Yaskawa INFORM job: test_long_tjr3.JBI

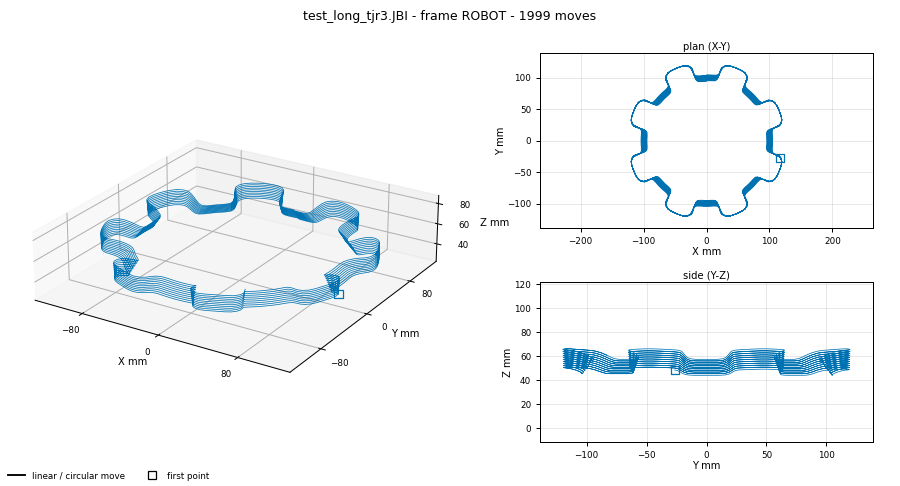
[picture p0: tool path of test_long_tjr3.JBI in frame ROBOT, 1999 of 2000 moves have a stored position in this frame; points joined in program order, loops and branches not executed]
version: 0
/JOB
//NAME test_long
//POS
///NPOS 48,0,0,2,0,0
///TOOL 1
///POSTYPE ROBOT
///RECTAN
///RCONF 1,0,0,0,0,0,0,0,0,0,0,0,0,0,0,0,0,0,0,0,0,0,0,0
C00000=118.780,-30.320,48.810,0.0300,0.0100,1.0000
C00001=116.910,-26.570,48.590,0.0400,0.0300,1.0000
C00002=114.000,-24.360,48.180,0.0300,0.0400,1.0000
C00003=110.720,-22.590,47.350,-0.0000,-0.0000,1.0000
C00004=107.770,-20.860,46.290,-0.0700,-0.1000,0.9900
C00005=105.620,-18.820,45.250,-0.2500,-0.2300,0.9400
C00006=104.550,-15.720,44.490,-0.5500,-0.1000,0.8300
C00007=104.610,-10.680,44.190,-0.6000,0.0300,0.8000
C00008=104.980,-5.420,44.180,-0.6000,0.0300,0.8000
C00009=105.130,0.000,44.190,-0.6000,0.0000,0.8000
C00010=104.980,5.420,44.180,-0.6000,-0.0300,0.8000
C00011=104.610,10.680,44.190,-0.6000,-0.0300,0.8000
C00012=104.550,15.720,44.490,-0.5500,0.1000,0.8300
C00013=105.620,18.820,45.250,-0.2500,0.2300,0.9400
C00014=107.770,20.860,46.290,-0.0700,0.1000,0.9900
C00015=110.720,22.590,47.350,-0.0000,0.0000,1.0000
C00016=114.000,24.360,48.180,0.0300,-0.0400,1.0000
C00017=116.910,26.570,48.590,0.0400,-0.0300,1.0000
C00018=118.780,30.320,48.810,0.0300,-0.0100,1.0000
C00019=119.290,35.170,48.990,0.0200,0.0000,1.0000
C00020=118.250,40.300,49.160,0.0000,0.0000,1.0000
C00021=116.480,45.340,49.280,0.0000,0.0000,1.0000
C00022=114.420,50.300,49.280,0.0000,0.0000,1.0000
C00023=112.110,55.120,49.160,0.0000,0.0000,1.0000
C00024=109.220,59.480,48.990,0.0200,0.0100,1.0000
C00025=105.430,62.550,48.810,0.0200,0.0300,1.0000
C00026=101.460,63.880,48.590,0.0000,0.0500,1.0000
C00027=97.840,63.390,48.180,-0.0100,0.0500,1.0000
C00028=94.260,62.320,47.350,0.0000,-0.0000,1.0000
C00029=90.960,61.450,46.290,0.0300,-0.1200,0.9900
C00030=87.990,61.380,45.250,-0.0200,-0.3400,0.9400
C00031=85.040,62.810,44.490,-0.3200,-0.4600,0.8300
C00032=81.530,66.420,44.190,-0.4500,-0.4000,0.8000
C00033=78.070,70.400,44.180,-0.4500,-0.4000,0.8000
C00034=74.330,74.330,44.190,-0.4300,-0.4300,0.8000
C00035=70.400,78.070,44.180,-0.4000,-0.4500,0.8000
C00036=66.420,81.530,44.190,-0.4000,-0.4500,0.8000
C00037=62.810,85.040,44.490,-0.4600,-0.3200,0.8300
C00038=61.380,87.990,45.250,-0.3400,-0.0200,0.9400
C00039=61.450,90.960,46.290,-0.1200,0.0300,0.9900
C00040=62.320,94.260,47.350,-0.0000,0.0000,1.0000
C00041=63.390,97.840,48.180,0.0500,-0.0100,1.0000
C00042=63.880,101.460,48.590,0.0500,0.0000,1.0000
C00043=62.550,105.430,48.810,0.0300,0.0200,1.0000
C00044=59.480,109.220,48.990,0.0100,0.0200,1.0000
C00045=55.120,112.110,49.160,0.0000,0.0000,1.0000
C00046=50.300,114.420,49.280,0.0000,0.0000,1.0000
C00047=45.340,116.480,49.280,0.0000,0.0000,1.0000
C00048=40.300,118.250,49.160,0.0000,0.0000,1.0000
C00049=35.170,119.290,48.990,0.0000,0.0200,1.0000
C00050=30.320,118.780,48.810,-0.0100,0.0300,1.0000
C00051=26.570,116.910,48.590,-0.0300,0.0400,1.0000
C00052=24.360,114.000,48.180,-0.0400,0.0300,1.0000
C00053=22.590,110.720,47.350,0.0000,-0.0000,1.0000
C00054=20.860,107.770,46.290,0.1000,-0.0700,0.9900
C00055=18.820,105.620,45.250,0.2300,-0.2500,0.9400
C00056=15.720,104.550,44.490,0.1000,-0.5500,0.8300
C00057=10.680,104.610,44.190,-0.0300,-0.6000,0.8000
C00058=5.420,104.980,44.180,-0.0300,-0.6000,0.8000
C00059=0.000,105.130,44.190,0.0000,-0.6000,0.8000
C00060=0.000,104.090,45.540,0.0000,-0.6100,0.7900
C00061=5.330,103.950,45.530,-0.0300,-0.6100,0.7900
C00062=10.520,103.590,45.540,-0.0300,-0.6100,0.7900
C00063=15.530,103.560,45.860,0.1100,-0.5500,0.8300
C00064=18.580,104.710,46.670,0.2300,-0.2300,0.9500
C00065=20.580,106.990,47.770,0.0900,-0.0500,0.9900
C00066=22.280,110.120,48.910,-0.0100,0.0000,1.0000
C00067=24.030,113.600,49.800,-0.0500,0.0300,1.0000
C00068=26.200,116.710,50.240,-0.0400,0.0500,1.0000
C00069=29.980,118.740,50.470,-0.0100,0.0300,1.0000
C00070=34.900,119.340,50.660,0.0000,0.0200,1.0000
C00071=40.120,118.310,50.850,0.0000,0.0000,1.0000
C00072=45.280,116.500,50.980,0.0000,0.0000,1.0000
C00073=50.360,114.400,50.980,0.0000,0.0000,1.0000
C00074=55.290,112.020,50.850,0.0000,0.0000,1.0000
C00075=59.710,109.060,50.660,0.0200,0.0200,1.0000
C00076=62.770,105.160,50.470,0.0300,0.0200,1.0000
C00077=64.000,101.050,50.240,0.0600,0.0000,1.0000
C00078=63.340,97.320,49.800,0.0600,-0.0200,1.0000
C00079=62.110,93.620,48.910,0.0100,-0.0000,1.0000
C00080=61.100,90.210,47.770,-0.1000,0.0300,0.9900
C00081=60.910,87.180,46.670,-0.3200,-0.0000,0.9500
C00082=62.250,84.200,45.860,-0.4700,-0.3100,0.8300
C00083=65.810,80.690,45.540,-0.4100,-0.4500,0.7900
C00084=69.740,77.270,45.530,-0.4100,-0.4500,0.7900
C00085=73.610,73.610,45.540,-0.4300,-0.4300,0.7900
C00086=77.270,69.740,45.530,-0.4500,-0.4100,0.7900
C00087=80.690,65.810,45.540,-0.4500,-0.4100,0.7900
C00088=84.200,62.250,45.860,-0.3100,-0.4700,0.8300
C00089=87.180,60.910,46.670,-0.0000,-0.3200,0.9500
C00090=90.210,61.100,47.770,0.0300,-0.1000,0.9900
C00091=93.620,62.110,48.910,-0.0000,0.0100,1.0000
C00092=97.320,63.340,49.800,-0.0200,0.0600,1.0000
C00093=101.050,64.000,50.240,0.0000,0.0600,1.0000
C00094=105.160,62.770,50.470,0.0200,0.0300,1.0000
C00095=109.060,59.710,50.660,0.0200,0.0200,1.0000
C00096=112.020,55.290,50.850,0.0000,0.0000,1.0000
C00097=114.400,50.360,50.980,0.0000,0.0000,1.0000
C00098=116.500,45.280,50.980,0.0000,0.0000,1.0000
C00099=118.310,40.120,50.850,0.0000,0.0000,1.0000
C00100=119.340,34.900,50.660,0.0200,0.0000,1.0000
C00101=118.740,29.980,50.470,0.0300,-0.0100,1.0000
C00102=116.710,26.200,50.240,0.0500,-0.0400,1.0000
C00103=113.600,24.030,49.800,0.0300,-0.0500,1.0000
C00104=110.120,22.280,48.910,0.0000,-0.0100,1.0000
C00105=106.990,20.580,47.770,-0.0500,0.0900,0.9900
C00106=104.710,18.580,46.670,-0.2300,0.2300,0.9500
C00107=103.560,15.530,45.860,-0.5500,0.1100,0.8300
C00108=103.590,10.520,45.540,-0.6100,-0.0300,0.7900
C00109=103.950,5.330,45.530,-0.6100,-0.0300,0.7900
C00110=104.090,0.000,45.540,-0.6100,0.0000,0.7900
C00111=103.950,-5.330,45.530,-0.6100,0.0300,0.7900
C00112=103.590,-10.520,45.540,-0.6100,0.0300,0.7900
C00113=103.560,-15.530,45.860,-0.5500,-0.1100,0.8300
C00114=104.710,-18.580,46.670,-0.2300,-0.2300,0.9500
C00115=106.990,-20.580,47.770,-0.0500,-0.0900,0.9900
C00116=110.120,-22.280,48.910,0.0000,0.0100,1.0000
C00117=113.600,-24.030,49.800,0.0300,0.0500,1.0000
C00118=116.710,-26.200,50.240,0.0500,0.0400,1.0000
C00119=118.740,-29.980,50.470,0.0300,0.0100,1.0000
C00120=119.340,-34.900,50.660,0.0200,-0.0000,1.0000
C00121=118.310,-40.120,50.850,0.0000,-0.0000,1.0000
C00122=116.500,-45.280,50.980,0.0000,-0.0000,1.0000
C00123=114.400,-50.360,50.980,0.0000,-0.0000,1.0000
C00124=112.020,-55.290,50.850,0.0000,-0.0000,1.0000
C00125=109.060,-59.710,50.660,0.0200,-0.0200,1.0000
C00126=105.160,-62.770,50.470,0.0200,-0.0300,1.0000
C00127=101.050,-64.000,50.240,0.0000,-0.0600,1.0000
C00128=97.320,-63.340,49.800,-0.0200,-0.0600,1.0000
C00129=93.620,-62.110,48.910,-0.0000,-0.0100,1.0000
C00130=90.210,-61.100,47.770,0.0300,0.1000,0.9900
C00131=87.180,-60.910,46.670,-0.0000,0.3200,0.9500
C00132=84.200,-62.250,45.860,-0.3100,0.4700,0.8300
C00133=80.690,-65.810,45.540,-0.4500,0.4100,0.7900
C00134=77.270,-69.740,45.530,-0.4500,0.4100,0.7900
C00135=73.610,-73.610,45.540,-0.4300,0.4300,0.7900
C00136=69.740,-77.270,45.530,-0.4100,0.4500,0.7900
C00137=65.810,-80.690,45.540,-0.4100,0.4500,0.7900
C00138=62.250,-84.200,45.860,-0.4700,0.3100,0.8300
C00139=60.910,-87.180,46.670,-0.3200,0.0000,0.9500
C00140=61.100,-90.210,47.770,-0.1000,-0.0300,0.9900
C00141=62.110,-93.620,48.910,0.0100,0.0000,1.0000
C00142=63.340,-97.320,49.800,0.0600,0.0200,1.0000
C00143=64.000,-101.050,50.240,0.0600,-0.0000,1.0000
C00144=62.770,-105.160,50.470,0.0300,-0.0200,1.0000
C00145=59.710,-109.060,50.660,0.0200,-0.0200,1.0000
C00146=55.290,-112.020,50.850,0.0000,-0.0000,1.0000
C00147=50.360,-114.400,50.980,0.0000,-0.0000,1.0000
C00148=45.280,-116.500,50.980,0.0000,-0.0000,1.0000
C00149=40.120,-118.310,50.850,0.0000,-0.0000,1.0000
C00150=34.900,-119.340,50.660,0.0000,-0.0200,1.0000
C00151=29.980,-118.740,50.470,-0.0100,-0.0300,1.0000
C00152=26.200,-116.710,50.240,-0.0400,-0.0500,1.0000
C00153=24.030,-113.600,49.800,-0.0500,-0.0300,1.0000
C00154=22.280,-110.120,48.910,-0.0100,-0.0000,1.0000
C00155=20.580,-106.990,47.770,0.0900,0.0500,0.9900
C00156=18.580,-104.710,46.670,0.2300,0.2300,0.9500
C00157=15.530,-103.560,45.860,0.1100,0.5500,0.8300
C00158=10.520,-103.590,45.540,-0.0300,0.6100,0.7900
C00159=5.330,-103.950,45.530,-0.0300,0.6100,0.7900
C00160=0.000,-104.090,45.540,0.0000,0.6100,0.7900
C00161=0.000,-104.090,45.540,0.0000,0.6100,0.7900
C00162=-5.330,-103.950,45.530,0.0300,0.6100,0.7900
C00163=-10.520,-103.590,45.540,0.0300,0.6100,0.7900
C00164=-15.530,-103.560,45.860,-0.1100,0.5500,0.8300
C00165=-18.580,-104.710,46.670,-0.2300,0.2300,0.9500
C00166=-20.580,-106.990,47.770,-0.0900,0.0500,0.9900
C00167=-22.280,-110.120,48.910,0.0100,-0.0000,1.0000
C00168=-24.030,-113.600,49.800,0.0500,-0.0300,1.0000
C00169=-26.200,-116.710,50.240,0.0400,-0.0500,1.0000
C00170=-29.980,-118.740,50.470,0.0100,-0.0300,1.0000
C00171=-34.900,-119.340,50.660,-0.0000,-0.0200,1.0000
C00172=-40.120,-118.310,50.850,-0.0000,-0.0000,1.0000
C00173=-45.280,-116.500,50.980,-0.0000,-0.0000,1.0000
C00174=-50.360,-114.400,50.980,-0.0000,-0.0000,1.0000
C00175=-55.290,-112.020,50.850,-0.0000,-0.0000,1.0000
C00176=-59.710,-109.060,50.660,-0.0200,-0.0200,1.0000
C00177=-62.770,-105.160,50.470,-0.0300,-0.0200,1.0000
C00178=-64.000,-101.050,50.240,-0.0600,-0.0000,1.0000
C00179=-63.340,-97.320,49.800,-0.0600,0.0200,1.0000
C00180=-62.110,-93.620,48.910,-0.0100,0.0000,1.0000
C00181=-61.100,-90.210,47.770,0.1000,-0.0300,0.9900
C00182=-60.910,-87.180,46.670,0.3200,0.0000,0.9500
C00183=-62.250,-84.200,45.860,0.4700,0.3100,0.8300
C00184=-65.810,-80.690,45.540,0.4100,0.4500,0.7900
C00185=-69.740,-77.270,45.530,0.4100,0.4500,0.7900
C00186=-73.610,-73.610,45.540,0.4300,0.4300,0.7900
C00187=-77.270,-69.740,45.530,0.4500,0.4100,0.7900
C00188=-80.690,-65.810,45.540,0.4500,0.4100,0.7900
C00189=-84.200,-62.250,45.860,0.3100,0.4700,0.8300
C00190=-87.180,-60.910,46.670,0.0000,0.3200,0.9500
C00191=-90.210,-61.100,47.770,-0.0300,0.1000,0.9900
C00192=-93.620,-62.110,48.910,0.0000,-0.0100,1.0000
C00193=-97.320,-63.340,49.800,0.0200,-0.0600,1.0000
C00194=-101.050,-64.000,50.240,-0.0000,-0.0600,1.0000
C00195=-105.160,-62.770,50.470,-0.0200,-0.0300,1.0000
C00196=-109.060,-59.710,50.660,-0.0200,-0.0200,1.0000
C00197=-112.020,-55.290,50.850,-0.0000,-0.0000,1.0000
C00198=-114.400,-50.360,50.980,-0.0000,-0.0000,1.0000
C00199=-116.500,-45.280,50.980,-0.0000,-0.0000,1.0000
C00200=-118.310,-40.120,50.850,-0.0000,-0.0000,1.0000
C00201=-119.340,-34.900,50.660,-0.0200,-0.0000,1.0000
C00202=-118.740,-29.980,50.470,-0.0300,0.0100,1.0000
C00203=-116.710,-26.200,50.240,-0.0500,0.0400,1.0000
C00204=-113.600,-24.030,49.800,-0.0300,0.0500,1.0000
C00205=-110.120,-22.280,48.910,-0.0000,0.0100,1.0000
C00206=-106.990,-20.580,47.770,0.0500,-0.0900,0.9900
C00207=-104.710,-18.580,46.670,0.2300,-0.2300,0.9500
C00208=-103.560,-15.530,45.860,0.5500,-0.1100,0.8300
C00209=-103.590,-10.520,45.540,0.6100,0.0300,0.7900
C00210=-103.950,-5.330,45.530,0.6100,0.0300,0.7900
C00211=-104.090,0.000,45.540,0.6100,-0.0000,0.7900
C00212=-103.950,5.330,45.530,0.6100,-0.0300,0.7900
C00213=-103.590,10.520,45.540,0.6100,-0.0300,0.7900
C00214=-103.560,15.530,45.860,0.5500,0.1100,0.8300
C00215=-104.710,18.580,46.670,0.2300,0.2300,0.9500
C00216=-106.990,20.580,47.770,0.0500,0.0900,0.9900
C00217=-110.120,22.280,48.910,-0.0000,-0.0100,1.0000
C00218=-113.600,24.030,49.800,-0.0300,-0.0500,1.0000
C00219=-116.710,26.200,50.240,-0.0500,-0.0400,1.0000
C00220=-118.740,29.980,50.470,-0.0300,-0.0100,1.0000
C00221=-119.340,34.900,50.660,-0.0200,0.0000,1.0000
C00222=-118.310,40.120,50.850,-0.0000,0.0000,1.0000
C00223=-116.500,45.280,50.980,-0.0000,0.0000,1.0000
C00224=-114.400,50.360,50.980,-0.0000,0.0000,1.0000
C00225=-112.020,55.290,50.850,-0.0000,0.0000,1.0000
C00226=-109.060,59.710,50.660,-0.0200,0.0200,1.0000
C00227=-105.160,62.770,50.470,-0.0200,0.0300,1.0000
C00228=-101.050,64.000,50.240,-0.0000,0.0600,1.0000
C00229=-97.320,63.340,49.800,0.0200,0.0600,1.0000
C00230=-93.620,62.110,48.910,0.0000,0.0100,1.0000
C00231=-90.210,61.100,47.770,-0.0300,-0.1000,0.9900
C00232=-87.180,60.910,46.670,0.0000,-0.3200,0.9500
C00233=-84.200,62.250,45.860,0.3100,-0.4700,0.8300
C00234=-80.690,65.810,45.540,0.4500,-0.4100,0.7900
C00235=-77.270,69.740,45.530,0.4500,-0.4100,0.7900
C00236=-73.610,73.610,45.540,0.4300,-0.4300,0.7900
C00237=-69.740,77.270,45.530,0.4100,-0.4500,0.7900
C00238=-65.810,80.690,45.540,0.4100,-0.4500,0.7900
C00239=-62.250,84.200,45.860,0.4700,-0.3100,0.8300
C00240=-60.910,87.180,46.670,0.3200,-0.0000,0.9500
C00241=-61.100,90.210,47.770,0.1000,0.0300,0.9900
C00242=-62.110,93.620,48.910,-0.0100,-0.0000,1.0000
C00243=-63.340,97.320,49.800,-0.0600,-0.0200,1.0000
C00244=-64.000,101.050,50.240,-0.0600,0.0000,1.0000
C00245=-62.770,105.160,50.470,-0.0300,0.0200,1.0000
C00246=-59.710,109.060,50.660,-0.0200,0.0200,1.0000
C00247=-55.290,112.020,50.850,-0.0000,0.0000,1.0000
C00248=-50.360,114.400,50.980,-0.0000,0.0000,1.0000
C00249=-45.280,116.500,50.980,-0.0000,0.0000,1.0000
C00250=-40.120,118.310,50.850,-0.0000,0.0000,1.0000
C00251=-34.900,119.340,50.660,-0.0000,0.0200,1.0000
C00252=-29.980,118.740,50.470,0.0100,0.0300,1.0000
C00253=-26.200,116.710,50.240,0.0400,0.0500,1.0000
C00254=-24.030,113.600,49.800,0.0500,0.0300,1.0000
C00255=-22.280,110.120,48.910,0.0100,0.0000,1.0000
C00256=-20.580,106.990,47.770,-0.0900,-0.0500,0.9900
C00257=-18.580,104.710,46.670,-0.2300,-0.2300,0.9500
C00258=-15.530,103.560,45.860,-0.1100,-0.5500,0.8300
C00259=-10.520,103.590,45.540,0.0300,-0.6100,0.7900
C00260=-5.330,103.950,45.530,0.0300,-0.6100,0.7900
C00261=0.000,104.090,45.540,0.0000,-0.6100,0.7900
C00262=0.000,103.050,46.880,0.0000,-0.6100,0.7900
C00263=-5.230,102.920,46.870,0.0300,-0.6100,0.7900
C00264=-10.360,102.570,46.890,0.0300,-0.6100,0.7900
C00265=-15.330,102.560,47.230,-0.1200,-0.5500,0.8200
C00266=-18.330,103.800,48.080,-0.2200,-0.2100,0.9500
C00267=-20.300,106.210,49.250,-0.0800,-0.0400,1.0000
C00268=-21.970,109.510,50.470,0.0200,0.0100,1.0000
C00269=-23.690,113.200,51.410,0.0600,0.0300,1.0000
C00270=-25.830,116.510,51.880,0.0500,0.0500,1.0000
C00271=-29.630,118.700,52.130,0.0100,0.0400,1.0000
C00272=-34.620,119.390,52.340,-0.0000,0.0300,1.0000
C00273=-39.940,118.360,52.540,-0.0000,0.0000,1.0000
C00274=-45.220,116.520,52.680,-0.0000,0.0000,1.0000
C00275=-50.420,114.370,52.680,-0.0000,0.0000,1.0000
C00276=-55.450,111.940,52.540,-0.0000,0.0000,1.0000
C00277=-59.940,108.900,52.340,-0.0200,0.0200,1.0000
C00278=-62.980,104.880,52.130,-0.0400,0.0200,1.0000
C00279=-64.120,100.650,51.880,-0.0700,0.0000,1.0000
C00280=-63.290,96.790,51.410,-0.0700,-0.0200,1.0000
C00281=-61.900,92.970,50.470,-0.0200,-0.0100,1.0000
C00282=-60.750,89.460,49.250,0.0900,0.0200,1.0000
C00283=-60.430,86.360,48.080,0.3100,0.0100,0.9500
C00284=-61.680,83.360,47.230,0.4800,-0.3100,0.8200
C00285=-65.200,79.850,46.890,0.4100,-0.4500,0.7900
C00286=-69.070,76.470,46.870,0.4100,-0.4600,0.7900
C00287=-72.870,72.870,46.880,0.4300,-0.4300,0.7900
C00288=-76.470,69.070,46.870,0.4600,-0.4100,0.7900
C00289=-79.850,65.200,46.890,0.4500,-0.4100,0.7900
C00290=-83.360,61.680,47.230,0.3100,-0.4800,0.8200
C00291=-86.360,60.430,48.080,-0.0100,-0.3100,0.9500
C00292=-89.460,60.750,49.250,-0.0200,-0.0900,1.0000
C00293=-92.970,61.900,50.470,0.0100,0.0200,1.0000
C00294=-96.790,63.290,51.410,0.0200,0.0700,1.0000
C00295=-100.650,64.120,51.880,-0.0000,0.0700,1.0000
C00296=-104.880,62.980,52.130,-0.0200,0.0400,1.0000
C00297=-108.900,59.940,52.340,-0.0200,0.0200,1.0000
C00298=-111.940,55.450,52.540,-0.0000,0.0000,1.0000
C00299=-114.370,50.420,52.680,-0.0000,0.0000,1.0000
C00300=-116.520,45.220,52.680,-0.0000,0.0000,1.0000
C00301=-118.360,39.940,52.540,-0.0000,0.0000,1.0000
C00302=-119.390,34.620,52.340,-0.0300,0.0000,1.0000
C00303=-118.700,29.630,52.130,-0.0400,-0.0100,1.0000
C00304=-116.510,25.830,51.880,-0.0500,-0.0500,1.0000
C00305=-113.200,23.690,51.410,-0.0300,-0.0600,1.0000
C00306=-109.510,21.970,50.470,-0.0100,-0.0200,1.0000
C00307=-106.210,20.300,49.250,0.0400,0.0800,1.0000
C00308=-103.800,18.330,48.080,0.2100,0.2200,0.9500
C00309=-102.560,15.330,47.230,0.5500,0.1200,0.8200
C00310=-102.570,10.360,46.890,0.6100,-0.0300,0.7900
C00311=-102.920,5.230,46.870,0.6100,-0.0300,0.7900
C00312=-103.050,0.000,46.880,0.6100,-0.0000,0.7900
C00313=-102.920,-5.230,46.870,0.6100,0.0300,0.7900
C00314=-102.570,-10.360,46.890,0.6100,0.0300,0.7900
C00315=-102.560,-15.330,47.230,0.5500,-0.1200,0.8200
C00316=-103.800,-18.330,48.080,0.2100,-0.2200,0.9500
C00317=-106.210,-20.300,49.250,0.0400,-0.0800,1.0000
C00318=-109.510,-21.970,50.470,-0.0100,0.0200,1.0000
C00319=-113.200,-23.690,51.410,-0.0300,0.0600,1.0000
C00320=-116.510,-25.830,51.880,-0.0500,0.0500,1.0000
C00321=-118.700,-29.630,52.130,-0.0400,0.0100,1.0000
C00322=-119.390,-34.620,52.340,-0.0300,-0.0000,1.0000
C00323=-118.360,-39.940,52.540,-0.0000,-0.0000,1.0000
C00324=-116.520,-45.220,52.680,-0.0000,-0.0000,1.0000
C00325=-114.370,-50.420,52.680,-0.0000,-0.0000,1.0000
C00326=-111.940,-55.450,52.540,-0.0000,-0.0000,1.0000
C00327=-108.900,-59.940,52.340,-0.0200,-0.0200,1.0000
C00328=-104.880,-62.980,52.130,-0.0200,-0.0400,1.0000
C00329=-100.650,-64.120,51.880,-0.0000,-0.0700,1.0000
C00330=-96.790,-63.290,51.410,0.0200,-0.0700,1.0000
C00331=-92.970,-61.900,50.470,0.0100,-0.0200,1.0000
C00332=-89.460,-60.750,49.250,-0.0200,0.0900,1.0000
C00333=-86.360,-60.430,48.080,-0.0100,0.3100,0.9500
C00334=-83.360,-61.680,47.230,0.3100,0.4800,0.8200
C00335=-79.850,-65.200,46.890,0.4500,0.4100,0.7900
C00336=-76.470,-69.070,46.870,0.4600,0.4100,0.7900
C00337=-72.870,-72.870,46.880,0.4300,0.4300,0.7900
C00338=-69.070,-76.470,46.870,0.4100,0.4600,0.7900
C00339=-65.200,-79.850,46.890,0.4100,0.4500,0.7900
C00340=-61.680,-83.360,47.230,0.4800,0.3100,0.8200
C00341=-60.430,-86.360,48.080,0.3100,-0.0100,0.9500
C00342=-60.750,-89.460,49.250,0.0900,-0.0200,1.0000
C00343=-61.900,-92.970,50.470,-0.0200,0.0100,1.0000
C00344=-63.290,-96.790,51.410,-0.0700,0.0200,1.0000
C00345=-64.120,-100.650,51.880,-0.0700,-0.0000,1.0000
C00346=-62.980,-104.880,52.130,-0.0400,-0.0200,1.0000
C00347=-59.940,-108.900,52.340,-0.0200,-0.0200,1.0000
C00348=-55.450,-111.940,52.540,-0.0000,-0.0000,1.0000
C00349=-50.420,-114.370,52.680,-0.0000,-0.0000,1.0000
C00350=-45.220,-116.520,52.680,-0.0000,-0.0000,1.0000
C00351=-39.940,-118.360,52.540,-0.0000,-0.0000,1.0000
C00352=-34.620,-119.390,52.340,-0.0000,-0.0300,1.0000
C00353=-29.630,-118.700,52.130,0.0100,-0.0400,1.0000
C00354=-25.830,-116.510,51.880,0.0500,-0.0500,1.0000
C00355=-23.690,-113.200,51.410,0.0600,-0.0300,1.0000
C00356=-21.970,-109.510,50.470,0.0200,-0.0100,1.0000
C00357=-20.300,-106.210,49.250,-0.0800,0.0400,1.0000
C00358=-18.330,-103.800,48.080,-0.2200,0.2100,0.9500
C00359=-15.330,-102.560,47.230,-0.1200,0.5500,0.8200
C00360=-10.360,-102.570,46.890,0.0300,0.6100,0.7900
C00361=-5.230,-102.920,46.870,0.0300,0.6100,0.7900
C00362=0.000,-103.050,46.880,0.0000,0.6100,0.7900
C00363=0.000,-103.050,46.880,0.0000,0.6100,0.7900
C00364=5.230,-102.920,46.870,-0.0300,0.6100,0.7900
C00365=10.360,-102.570,46.890,-0.0300,0.6100,0.7900
C00366=15.330,-102.560,47.230,0.1200,0.5500,0.8200
C00367=18.330,-103.800,48.080,0.2200,0.2100,0.9500
C00368=20.300,-106.210,49.250,0.0800,0.0400,1.0000
C00369=21.970,-109.510,50.470,-0.0200,-0.0100,1.0000
C00370=23.690,-113.200,51.410,-0.0600,-0.0300,1.0000
C00371=25.830,-116.510,51.880,-0.0500,-0.0500,1.0000
C00372=29.630,-118.700,52.130,-0.0100,-0.0400,1.0000
C00373=34.620,-119.390,52.340,0.0000,-0.0300,1.0000
C00374=39.940,-118.360,52.540,0.0000,-0.0000,1.0000
C00375=45.220,-116.520,52.680,0.0000,-0.0000,1.0000
C00376=50.420,-114.370,52.680,0.0000,-0.0000,1.0000
C00377=55.450,-111.940,52.540,0.0000,-0.0000,1.0000
C00378=59.940,-108.900,52.340,0.0200,-0.0200,1.0000
C00379=62.980,-104.880,52.130,0.0400,-0.0200,1.0000
C00380=64.120,-100.650,51.880,0.0700,-0.0000,1.0000
C00381=63.290,-96.790,51.410,0.0700,0.0200,1.0000
C00382=61.900,-92.970,50.470,0.0200,0.0100,1.0000
C00383=60.750,-89.460,49.250,-0.0900,-0.0200,1.0000
C00384=60.430,-86.360,48.080,-0.3100,-0.0100,0.9500
C00385=61.680,-83.360,47.230,-0.4800,0.3100,0.8200
C00386=65.200,-79.850,46.890,-0.4100,0.4500,0.7900
C00387=69.070,-76.470,46.870,-0.4100,0.4600,0.7900
C00388=72.870,-72.870,46.880,-0.4300,0.4300,0.7900
C00389=76.470,-69.070,46.870,-0.4600,0.4100,0.7900
C00390=79.850,-65.200,46.890,-0.4500,0.4100,0.7900
C00391=83.360,-61.680,47.230,-0.3100,0.4800,0.8200
C00392=86.360,-60.430,48.080,0.0100,0.3100,0.9500
C00393=89.460,-60.750,49.250,0.0200,0.0900,1.0000
C00394=92.970,-61.900,50.470,-0.0100,-0.0200,1.0000
C00395=96.790,-63.290,51.410,-0.0200,-0.0700,1.0000
C00396=100.650,-64.120,51.880,0.0000,-0.0700,1.0000
C00397=104.880,-62.980,52.130,0.0200,-0.0400,1.0000
C00398=108.900,-59.940,52.340,0.0200,-0.0200,1.0000
C00399=111.940,-55.450,52.540,0.0000,-0.0000,1.0000
C00400=114.370,-50.420,52.680,0.0000,-0.0000,1.0000
C00401=116.520,-45.220,52.680,0.0000,-0.0000,1.0000
C00402=118.360,-39.940,52.540,0.0000,-0.0000,1.0000
C00403=119.390,-34.620,52.340,0.0300,-0.0000,1.0000
C00404=118.700,-29.630,52.130,0.0400,0.0100,1.0000
C00405=116.510,-25.830,51.880,0.0500,0.0500,1.0000
C00406=113.200,-23.690,51.410,0.0300,0.0600,1.0000
C00407=109.510,-21.970,50.470,0.0100,0.0200,1.0000
C00408=106.210,-20.300,49.250,-0.0400,-0.0800,1.0000
C00409=103.800,-18.330,48.080,-0.2100,-0.2200,0.9500
C00410=102.560,-15.330,47.230,-0.5500,-0.1200,0.8200
C00411=102.570,-10.360,46.890,-0.6100,0.0300,0.7900
C00412=102.920,-5.230,46.870,-0.6100,0.0300,0.7900
C00413=103.050,0.000,46.880,-0.6100,0.0000,0.7900
C00414=102.920,5.230,46.870,-0.6100,-0.0300,0.7900
C00415=102.570,10.360,46.890,-0.6100,-0.0300,0.7900
C00416=102.560,15.330,47.230,-0.5500,0.1200,0.8200
C00417=103.800,18.330,48.080,-0.2100,0.2200,0.9500
C00418=106.210,20.300,49.250,-0.0400,0.0800,1.0000
C00419=109.510,21.970,50.470,0.0100,-0.0200,1.0000
C00420=113.200,23.690,51.410,0.0300,-0.0600,1.0000
C00421=116.510,25.830,51.880,0.0500,-0.0500,1.0000
C00422=118.700,29.630,52.130,0.0400,-0.0100,1.0000
C00423=119.390,34.620,52.340,0.0300,0.0000,1.0000
C00424=118.360,39.940,52.540,0.0000,0.0000,1.0000
C00425=116.520,45.220,52.680,0.0000,0.0000,1.0000
C00426=114.370,50.420,52.680,0.0000,0.0000,1.0000
C00427=111.940,55.450,52.540,0.0000,0.0000,1.0000
C00428=108.900,59.940,52.340,0.0200,0.0200,1.0000
C00429=104.880,62.980,52.130,0.0200,0.0400,1.0000
C00430=100.650,64.120,51.880,0.0000,0.0700,1.0000
C00431=96.790,63.290,51.410,-0.0200,0.0700,1.0000
C00432=92.970,61.900,50.470,-0.0100,0.0200,1.0000
C00433=89.460,60.750,49.250,0.0200,-0.0900,1.0000
C00434=86.360,60.430,48.080,0.0100,-0.3100,0.9500
C00435=83.360,61.680,47.230,-0.3100,-0.4800,0.8200
C00436=79.850,65.200,46.890,-0.4500,-0.4100,0.7900
C00437=76.470,69.070,46.870,-0.4600,-0.4100,0.7900
C00438=72.870,72.870,46.880,-0.4300,-0.4300,0.7900
C00439=69.070,76.470,46.870,-0.4100,-0.4600,0.7900
C00440=65.200,79.850,46.890,-0.4100,-0.4500,0.7900
C00441=61.680,83.360,47.230,-0.4800,-0.3100,0.8200
C00442=60.430,86.360,48.080,-0.3100,0.0100,0.9500
C00443=60.750,89.460,49.250,-0.0900,0.0200,1.0000
C00444=61.900,92.970,50.470,0.0200,-0.0100,1.0000
C00445=63.290,96.790,51.410,0.0700,-0.0200,1.0000
C00446=64.120,100.650,51.880,0.0700,0.0000,1.0000
C00447=62.980,104.880,52.130,0.0400,0.0200,1.0000
C00448=59.940,108.900,52.340,0.0200,0.0200,1.0000
C00449=55.450,111.940,52.540,0.0000,0.0000,1.0000
C00450=50.420,114.370,52.680,0.0000,0.0000,1.0000
C00451=45.220,116.520,52.680,0.0000,0.0000,1.0000
C00452=39.940,118.360,52.540,0.0000,0.0000,1.0000
C00453=34.620,119.390,52.340,0.0000,0.0300,1.0000
C00454=29.630,118.700,52.130,-0.0100,0.0400,1.0000
C00455=25.830,116.510,51.880,-0.0500,0.0500,1.0000
C00456=23.690,113.200,51.410,-0.0600,0.0300,1.0000
C00457=21.970,109.510,50.470,-0.0200,0.0100,1.0000
C00458=20.300,106.210,49.250,0.0800,-0.0400,1.0000
C00459=18.330,103.800,48.080,0.2200,-0.2100,0.9500
C00460=15.330,102.560,47.230,0.1200,-0.5500,0.8200
C00461=10.360,102.570,46.890,-0.0300,-0.6100,0.7900
C00462=5.230,102.920,46.870,-0.0300,-0.6100,0.7900
C00463=0.000,103.050,46.880,0.0000,-0.6100,0.7900
C00464=0.000,102.010,48.220,0.0000,-0.6200,0.7900
C00465=5.140,101.870,48.210,-0.0300,-0.6200,0.7900
C00466=10.200,101.530,48.230,-0.0300,-0.6100,0.7900
C00467=15.130,101.560,48.590,0.1300,-0.5500,0.8200
C00468=18.090,102.880,49.490,0.2200,-0.1900,0.9600
C00469=20.020,105.420,50.730,0.0700,-0.0400,1.0000
C00470=21.650,108.900,52.030,-0.0300,0.0100,1.0000
C00471=23.350,112.790,53.030,-0.0700,0.0300,1.0000
C00472=25.460,116.310,53.530,-0.0600,0.0500,1.0000
C00473=29.270,118.660,53.800,-0.0100,0.0400,1.0000
C00474=34.340,119.440,54.010,0.0000,0.0300,1.0000
C00475=39.770,118.420,54.230,0.0000,0.0000,1.0000
C00476=45.160,116.550,54.380,0.0000,0.0000,1.0000
C00477=50.480,114.340,54.380,0.0000,0.0000,1.0000
C00478=55.620,111.860,54.230,0.0000,0.0000,1.0000
C00479=60.180,108.740,54.010,0.0200,0.0200,1.0000
C00480=63.200,104.600,53.800,0.0400,0.0200,1.0000
C00481=64.240,100.240,53.530,0.0800,-0.0000,1.0000
C00482=63.250,96.260,53.030,0.0800,-0.0300,1.0000
C00483=61.690,92.310,52.030,0.0300,-0.0100,1.0000
C00484=60.390,88.700,50.730,-0.0700,0.0200,1.0000
C00485=59.950,85.540,49.490,-0.2900,0.0200,0.9600
C00486=61.110,82.510,48.590,-0.4800,-0.3000,0.8200
C00487=64.580,79.010,48.230,-0.4200,-0.4500,0.7900
C00488=68.400,75.670,48.210,-0.4100,-0.4600,0.7900
C00489=72.130,72.130,48.220,-0.4400,-0.4400,0.7900
C00490=75.670,68.400,48.210,-0.4600,-0.4100,0.7900
C00491=79.010,64.580,48.230,-0.4500,-0.4200,0.7900
C00492=82.510,61.110,48.590,-0.3000,-0.4800,0.8200
C00493=85.540,59.950,49.490,0.0200,-0.2900,0.9600
C00494=88.700,60.390,50.730,0.0200,-0.0700,1.0000
C00495=92.310,61.690,52.030,-0.0100,0.0300,1.0000
C00496=96.260,63.250,53.030,-0.0300,0.0800,1.0000
C00497=100.240,64.240,53.530,-0.0000,0.0800,1.0000
C00498=104.600,63.200,53.800,0.0200,0.0400,1.0000
C00499=108.740,60.180,54.010,0.0200,0.0200,1.0000
C00500=111.860,55.620,54.230,0.0000,0.0000,1.0000
C00501=114.340,50.480,54.380,0.0000,0.0000,1.0000
C00502=116.550,45.160,54.380,0.0000,0.0000,1.0000
C00503=118.420,39.770,54.230,0.0000,0.0000,1.0000
C00504=119.440,34.340,54.010,0.0300,0.0000,1.0000
C00505=118.660,29.270,53.800,0.0400,-0.0100,1.0000
C00506=116.310,25.460,53.530,0.0500,-0.0600,1.0000
C00507=112.790,23.350,53.030,0.0300,-0.0700,1.0000
C00508=108.900,21.650,52.030,0.0100,-0.0300,1.0000
C00509=105.420,20.020,50.730,-0.0400,0.0700,1.0000
C00510=102.880,18.090,49.490,-0.1900,0.2200,0.9600
C00511=101.560,15.130,48.590,-0.5500,0.1300,0.8200
C00512=101.530,10.200,48.230,-0.6100,-0.0300,0.7900
C00513=101.870,5.140,48.210,-0.6200,-0.0300,0.7900
C00514=102.010,0.000,48.220,-0.6200,0.0000,0.7900
C00515=101.870,-5.140,48.210,-0.6200,0.0300,0.7900
C00516=101.530,-10.200,48.230,-0.6100,0.0300,0.7900
C00517=101.560,-15.130,48.590,-0.5500,-0.1300,0.8200
C00518=102.880,-18.090,49.490,-0.1900,-0.2200,0.9600
C00519=105.420,-20.020,50.730,-0.0400,-0.0700,1.0000
C00520=108.900,-21.650,52.030,0.0100,0.0300,1.0000
C00521=112.790,-23.350,53.030,0.0300,0.0700,1.0000
C00522=116.310,-25.460,53.530,0.0500,0.0600,1.0000
C00523=118.660,-29.270,53.800,0.0400,0.0100,1.0000
C00524=119.440,-34.340,54.010,0.0300,-0.0000,1.0000
C00525=118.420,-39.770,54.230,0.0000,-0.0000,1.0000
C00526=116.550,-45.160,54.380,0.0000,-0.0000,1.0000
C00527=114.340,-50.480,54.380,0.0000,-0.0000,1.0000
C00528=111.860,-55.620,54.230,0.0000,-0.0000,1.0000
C00529=108.740,-60.180,54.010,0.0200,-0.0200,1.0000
C00530=104.600,-63.200,53.800,0.0200,-0.0400,1.0000
C00531=100.240,-64.240,53.530,-0.0000,-0.0800,1.0000
C00532=96.260,-63.250,53.030,-0.0300,-0.0800,1.0000
C00533=92.310,-61.690,52.030,-0.0100,-0.0300,1.0000
C00534=88.700,-60.390,50.730,0.0200,0.0700,1.0000
C00535=85.540,-59.950,49.490,0.0200,0.2900,0.9600
C00536=82.510,-61.110,48.590,-0.3000,0.4800,0.8200
C00537=79.010,-64.580,48.230,-0.4500,0.4200,0.7900
C00538=75.670,-68.400,48.210,-0.4600,0.4100,0.7900
C00539=72.130,-72.130,48.220,-0.4400,0.4400,0.7900
C00540=68.400,-75.670,48.210,-0.4100,0.4600,0.7900
C00541=64.580,-79.010,48.230,-0.4200,0.4500,0.7900
C00542=61.110,-82.510,48.590,-0.4800,0.3000,0.8200
C00543=59.950,-85.540,49.490,-0.2900,-0.0200,0.9600
C00544=60.390,-88.700,50.730,-0.0700,-0.0200,1.0000
C00545=61.690,-92.310,52.030,0.0300,0.0100,1.0000
C00546=63.250,-96.260,53.030,0.0800,0.0300,1.0000
C00547=64.240,-100.240,53.530,0.0800,0.0000,1.0000
C00548=63.200,-104.600,53.800,0.0400,-0.0200,1.0000
C00549=60.180,-108.740,54.010,0.0200,-0.0200,1.0000
C00550=55.620,-111.860,54.230,0.0000,-0.0000,1.0000
C00551=50.480,-114.340,54.380,0.0000,-0.0000,1.0000
C00552=45.160,-116.550,54.380,0.0000,-0.0000,1.0000
C00553=39.770,-118.420,54.230,0.0000,-0.0000,1.0000
C00554=34.340,-119.440,54.010,0.0000,-0.0300,1.0000
C00555=29.270,-118.660,53.800,-0.0100,-0.0400,1.0000
C00556=25.460,-116.310,53.530,-0.0600,-0.0500,1.0000
C00557=23.350,-112.790,53.030,-0.0700,-0.0300,1.0000
C00558=21.650,-108.900,52.030,-0.0300,-0.0100,1.0000
C00559=20.020,-105.420,50.730,0.0700,0.0400,1.0000
C00560=18.090,-102.880,49.490,0.2200,0.1900,0.9600
C00561=15.130,-101.560,48.590,0.1300,0.5500,0.8200
C00562=10.200,-101.530,48.230,-0.0300,0.6100,0.7900
C00563=5.140,-101.870,48.210,-0.0300,0.6200,0.7900
C00564=0.000,-102.010,48.220,0.0000,0.6200,0.7900
C00565=0.000,-102.010,48.220,0.0000,0.6200,0.7900
C00566=-5.140,-101.870,48.210,0.0300,0.6200,0.7900
C00567=-10.200,-101.530,48.230,0.0300,0.6100,0.7900
C00568=-15.130,-101.560,48.590,-0.1300,0.5500,0.8200
C00569=-18.090,-102.880,49.490,-0.2200,0.1900,0.9600
C00570=-20.020,-105.420,50.730,-0.0700,0.0400,1.0000
C00571=-21.650,-108.900,52.030,0.0300,-0.0100,1.0000
C00572=-23.350,-112.790,53.030,0.0700,-0.0300,1.0000
C00573=-25.460,-116.310,53.530,0.0600,-0.0500,1.0000
C00574=-29.270,-118.660,53.800,0.0100,-0.0400,1.0000
C00575=-34.340,-119.440,54.010,-0.0000,-0.0300,1.0000
C00576=-39.770,-118.420,54.230,-0.0000,-0.0000,1.0000
C00577=-45.160,-116.550,54.380,-0.0000,-0.0000,1.0000
C00578=-50.480,-114.340,54.380,-0.0000,-0.0000,1.0000
C00579=-55.620,-111.860,54.230,-0.0000,-0.0000,1.0000
C00580=-60.180,-108.740,54.010,-0.0200,-0.0200,1.0000
C00581=-63.200,-104.600,53.800,-0.0400,-0.0200,1.0000
C00582=-64.240,-100.240,53.530,-0.0800,0.0000,1.0000
C00583=-63.250,-96.260,53.030,-0.0800,0.0300,1.0000
C00584=-61.690,-92.310,52.030,-0.0300,0.0100,1.0000
C00585=-60.390,-88.700,50.730,0.0700,-0.0200,1.0000
C00586=-59.950,-85.540,49.490,0.2900,-0.0200,0.9600
C00587=-61.110,-82.510,48.590,0.4800,0.3000,0.8200
C00588=-64.580,-79.010,48.230,0.4200,0.4500,0.7900
C00589=-68.400,-75.670,48.210,0.4100,0.4600,0.7900
C00590=-72.130,-72.130,48.220,0.4400,0.4400,0.7900
C00591=-75.670,-68.400,48.210,0.4600,0.4100,0.7900
C00592=-79.010,-64.580,48.230,0.4500,0.4200,0.7900
C00593=-82.510,-61.110,48.590,0.3000,0.4800,0.8200
C00594=-85.540,-59.950,49.490,-0.0200,0.2900,0.9600
C00595=-88.700,-60.390,50.730,-0.0200,0.0700,1.0000
C00596=-92.310,-61.690,52.030,0.0100,-0.0300,1.0000
C00597=-96.260,-63.250,53.030,0.0300,-0.0800,1.0000
C00598=-100.240,-64.240,53.530,0.0000,-0.0800,1.0000
C00599=-104.600,-63.200,53.800,-0.0200,-0.0400,1.0000
C00600=-108.740,-60.180,54.010,-0.0200,-0.0200,1.0000
C00601=-111.860,-55.620,54.230,-0.0000,-0.0000,1.0000
C00602=-114.340,-50.480,54.380,-0.0000,-0.0000,1.0000
C00603=-116.550,-45.160,54.380,-0.0000,-0.0000,1.0000
C00604=-118.420,-39.770,54.230,-0.0000,-0.0000,1.0000
C00605=-119.440,-34.340,54.010,-0.0300,-0.0000,1.0000
C00606=-118.660,-29.270,53.800,-0.0400,0.0100,1.0000
C00607=-116.310,-25.460,53.530,-0.0500,0.0600,1.0000
C00608=-112.790,-23.350,53.030,-0.0300,0.0700,1.0000
C00609=-108.900,-21.650,52.030,-0.0100,0.0300,1.0000
C00610=-105.420,-20.020,50.730,0.0400,-0.0700,1.0000
C00611=-102.880,-18.090,49.490,0.1900,-0.2200,0.9600
C00612=-101.560,-15.130,48.590,0.5500,-0.1300,0.8200
C00613=-101.530,-10.200,48.230,0.6100,0.0300,0.7900
C00614=-101.870,-5.140,48.210,0.6200,0.0300,0.7900
C00615=-102.010,0.000,48.220,0.6200,-0.0000,0.7900
C00616=-101.870,5.140,48.210,0.6200,-0.0300,0.7900
C00617=-101.530,10.200,48.230,0.6100,-0.0300,0.7900
C00618=-101.560,15.130,48.590,0.5500,0.1300,0.8200
C00619=-102.880,18.090,49.490,0.1900,0.2200,0.9600
C00620=-105.420,20.020,50.730,0.0400,0.0700,1.0000
C00621=-108.900,21.650,52.030,-0.0100,-0.0300,1.0000
C00622=-112.790,23.350,53.030,-0.0300,-0.0700,1.0000
C00623=-116.310,25.460,53.530,-0.0500,-0.0600,1.0000
C00624=-118.660,29.270,53.800,-0.0400,-0.0100,1.0000
C00625=-119.440,34.340,54.010,-0.0300,0.0000,1.0000
C00626=-118.420,39.770,54.230,-0.0000,0.0000,1.0000
C00627=-116.550,45.160,54.380,-0.0000,0.0000,1.0000
C00628=-114.340,50.480,54.380,-0.0000,0.0000,1.0000
C00629=-111.860,55.620,54.230,-0.0000,0.0000,1.0000
C00630=-108.740,60.180,54.010,-0.0200,0.0200,1.0000
C00631=-104.600,63.200,53.800,-0.0200,0.0400,1.0000
C00632=-100.240,64.240,53.530,0.0000,0.0800,1.0000
C00633=-96.260,63.250,53.030,0.0300,0.0800,1.0000
C00634=-92.310,61.690,52.030,0.0100,0.0300,1.0000
C00635=-88.700,60.390,50.730,-0.0200,-0.0700,1.0000
C00636=-85.540,59.950,49.490,-0.0200,-0.2900,0.9600
C00637=-82.510,61.110,48.590,0.3000,-0.4800,0.8200
C00638=-79.010,64.580,48.230,0.4500,-0.4200,0.7900
C00639=-75.670,68.400,48.210,0.4600,-0.4100,0.7900
C00640=-72.130,72.130,48.220,0.4400,-0.4400,0.7900
C00641=-68.400,75.670,48.210,0.4100,-0.4600,0.7900
C00642=-64.580,79.010,48.230,0.4200,-0.4500,0.7900
C00643=-61.110,82.510,48.590,0.4800,-0.3000,0.8200
C00644=-59.950,85.540,49.490,0.2900,0.0200,0.9600
C00645=-60.390,88.700,50.730,0.0700,0.0200,1.0000
C00646=-61.690,92.310,52.030,-0.0300,-0.0100,1.0000
C00647=-63.250,96.260,53.030,-0.0800,-0.0300,1.0000
C00648=-64.240,100.240,53.530,-0.0800,-0.0000,1.0000
C00649=-63.200,104.600,53.800,-0.0400,0.0200,1.0000
C00650=-60.180,108.740,54.010,-0.0200,0.0200,1.0000
C00651=-55.620,111.860,54.230,-0.0000,0.0000,1.0000
C00652=-50.480,114.340,54.380,-0.0000,0.0000,1.0000
C00653=-45.160,116.550,54.380,-0.0000,0.0000,1.0000
C00654=-39.770,118.420,54.230,-0.0000,0.0000,1.0000
C00655=-34.340,119.440,54.010,-0.0000,0.0300,1.0000
C00656=-29.270,118.660,53.800,0.0100,0.0400,1.0000
C00657=-25.460,116.310,53.530,0.0600,0.0500,1.0000
C00658=-23.350,112.790,53.030,0.0700,0.0300,1.0000
C00659=-21.650,108.900,52.030,0.0300,0.0100,1.0000
C00660=-20.020,105.420,50.730,-0.0700,-0.0400,1.0000
C00661=-18.090,102.880,49.490,-0.2200,-0.1900,0.9600
C00662=-15.130,101.560,48.590,-0.1300,-0.5500,0.8200
C00663=-10.200,101.530,48.230,0.0300,-0.6100,0.7900
C00664=-5.140,101.870,48.210,0.0300,-0.6200,0.7900
C00665=0.000,102.010,48.220,0.0000,-0.6200,0.7900
C00666=0.000,100.950,49.560,0.0000,-0.6200,0.7800
C00667=-5.040,100.820,49.550,0.0300,-0.6200,0.7800
C00668=-10.040,100.490,49.560,0.0200,-0.6200,0.7900
C00669=-14.930,100.550,49.940,-0.1400,-0.5500,0.8200
C00670=-17.840,101.950,50.890,-0.2100,-0.1700,0.9600
C00671=-19.730,104.630,52.210,-0.0600,-0.0300,1.0000
C00672=-21.340,108.280,53.580,0.0300,0.0100,1.0000
C00673=-23.000,112.380,54.640,0.0800,0.0400,1.0000
C00674=-25.080,116.100,55.180,0.0700,0.0600,1.0000
C00675=-28.920,118.610,55.460,0.0200,0.0500,1.0000
C00676=-34.050,119.490,55.690,-0.0000,0.0300,1.0000
C00677=-39.590,118.480,55.920,-0.0000,0.0000,1.0000
C00678=-45.100,116.570,56.080,-0.0000,0.0000,1.0000
C00679=-50.540,114.320,56.080,-0.0000,0.0000,1.0000
C00680=-55.790,111.770,55.920,-0.0000,0.0000,1.0000
C00681=-60.410,108.570,55.690,-0.0200,0.0200,1.0000
C00682=-63.430,104.320,55.460,-0.0500,0.0200,1.0000
C00683=-64.360,99.830,55.180,-0.0900,-0.0100,1.0000
C00684=-63.200,95.730,54.640,-0.0800,-0.0300,1.0000
C00685=-61.480,91.650,53.580,-0.0300,-0.0100,1.0000
C00686=-60.030,87.930,52.210,0.0600,0.0200,1.0000
C00687=-59.470,84.710,50.890,0.2700,0.0300,0.9600
C00688=-60.540,81.660,49.940,0.4900,-0.2900,0.8200
C00689=-63.960,78.160,49.560,0.4200,-0.4500,0.7900
C00690=-67.730,74.860,49.550,0.4100,-0.4600,0.7800
C00691=-71.380,71.380,49.560,0.4400,-0.4400,0.7800
C00692=-74.860,67.730,49.550,0.4600,-0.4100,0.7800
C00693=-78.160,63.960,49.560,0.4500,-0.4200,0.7900
C00694=-81.660,60.540,49.940,0.2900,-0.4900,0.8200
C00695=-84.710,59.470,50.890,-0.0300,-0.2700,0.9600
C00696=-87.930,60.030,52.210,-0.0200,-0.0600,1.0000
C00697=-91.650,61.480,53.580,0.0100,0.0300,1.0000
C00698=-95.730,63.200,54.640,0.0300,0.0800,1.0000
C00699=-99.830,64.360,55.180,0.0100,0.0900,1.0000
C00700=-104.320,63.430,55.460,-0.0200,0.0500,1.0000
C00701=-108.570,60.410,55.690,-0.0200,0.0200,1.0000
C00702=-111.770,55.790,55.920,-0.0000,0.0000,1.0000
C00703=-114.320,50.540,56.080,-0.0000,0.0000,1.0000
C00704=-116.570,45.100,56.080,-0.0000,0.0000,1.0000
C00705=-118.480,39.590,55.920,-0.0000,0.0000,1.0000
C00706=-119.490,34.050,55.690,-0.0300,0.0000,1.0000
C00707=-118.610,28.920,55.460,-0.0500,-0.0200,1.0000
C00708=-116.100,25.080,55.180,-0.0600,-0.0700,1.0000
C00709=-112.380,23.000,54.640,-0.0400,-0.0800,1.0000
C00710=-108.280,21.340,53.580,-0.0100,-0.0300,1.0000
C00711=-104.630,19.730,52.210,0.0300,0.0600,1.0000
C00712=-101.950,17.840,50.890,0.1700,0.2100,0.9600
C00713=-100.550,14.930,49.940,0.5500,0.1400,0.8200
C00714=-100.490,10.040,49.560,0.6200,-0.0200,0.7900
C00715=-100.820,5.040,49.550,0.6200,-0.0300,0.7800
C00716=-100.950,0.000,49.560,0.6200,-0.0000,0.7800
C00717=-100.820,-5.040,49.550,0.6200,0.0300,0.7800
C00718=-100.490,-10.040,49.560,0.6200,0.0200,0.7900
C00719=-100.550,-14.930,49.940,0.5500,-0.1400,0.8200
C00720=-101.950,-17.840,50.890,0.1700,-0.2100,0.9600
C00721=-104.630,-19.730,52.210,0.0300,-0.0600,1.0000
C00722=-108.280,-21.340,53.580,-0.0100,0.0300,1.0000
C00723=-112.380,-23.000,54.640,-0.0400,0.0800,1.0000
C00724=-116.100,-25.080,55.180,-0.0600,0.0700,1.0000
C00725=-118.610,-28.920,55.460,-0.0500,0.0200,1.0000
C00726=-119.490,-34.050,55.690,-0.0300,-0.0000,1.0000
C00727=-118.480,-39.590,55.920,-0.0000,-0.0000,1.0000
C00728=-116.570,-45.100,56.080,-0.0000,-0.0000,1.0000
C00729=-114.320,-50.540,56.080,-0.0000,-0.0000,1.0000
C00730=-111.770,-55.790,55.920,-0.0000,-0.0000,1.0000
C00731=-108.570,-60.410,55.690,-0.0200,-0.0200,1.0000
C00732=-104.320,-63.430,55.460,-0.0200,-0.0500,1.0000
C00733=-99.830,-64.360,55.180,0.0100,-0.0900,1.0000
C00734=-95.730,-63.200,54.640,0.0300,-0.0800,1.0000
C00735=-91.650,-61.480,53.580,0.0100,-0.0300,1.0000
C00736=-87.930,-60.030,52.210,-0.0200,0.0600,1.0000
C00737=-84.710,-59.470,50.890,-0.0300,0.2700,0.9600
C00738=-81.660,-60.540,49.940,0.2900,0.4900,0.8200
C00739=-78.160,-63.960,49.560,0.4500,0.4200,0.7900
C00740=-74.860,-67.730,49.550,0.4600,0.4100,0.7800
C00741=-71.380,-71.380,49.560,0.4400,0.4400,0.7800
C00742=-67.730,-74.860,49.550,0.4100,0.4600,0.7800
C00743=-63.960,-78.160,49.560,0.4200,0.4500,0.7900
C00744=-60.540,-81.660,49.940,0.4900,0.2900,0.8200
C00745=-59.470,-84.710,50.890,0.2700,-0.0300,0.9600
C00746=-60.030,-87.930,52.210,0.0600,-0.0200,1.0000
C00747=-61.480,-91.650,53.580,-0.0300,0.0100,1.0000
C00748=-63.200,-95.730,54.640,-0.0800,0.0300,1.0000
C00749=-64.360,-99.830,55.180,-0.0900,0.0100,1.0000
C00750=-63.430,-104.320,55.460,-0.0500,-0.0200,1.0000
C00751=-60.410,-108.570,55.690,-0.0200,-0.0200,1.0000
C00752=-55.790,-111.770,55.920,-0.0000,-0.0000,1.0000
C00753=-50.540,-114.320,56.080,-0.0000,-0.0000,1.0000
C00754=-45.100,-116.570,56.080,-0.0000,-0.0000,1.0000
C00755=-39.590,-118.480,55.920,-0.0000,-0.0000,1.0000
C00756=-34.050,-119.490,55.690,-0.0000,-0.0300,1.0000
C00757=-28.920,-118.610,55.460,0.0200,-0.0500,1.0000
C00758=-25.080,-116.100,55.180,0.0700,-0.0600,1.0000
C00759=-23.000,-112.380,54.640,0.0800,-0.0400,1.0000
C00760=-21.340,-108.280,53.580,0.0300,-0.0100,1.0000
C00761=-19.730,-104.630,52.210,-0.0600,0.0300,1.0000
C00762=-17.840,-101.950,50.890,-0.2100,0.1700,0.9600
C00763=-14.930,-100.550,49.940,-0.1400,0.5500,0.8200
C00764=-10.040,-100.490,49.560,0.0200,0.6200,0.7900
C00765=-5.040,-100.820,49.550,0.0300,0.6200,0.7800
C00766=0.000,-100.950,49.560,0.0000,0.6200,0.7800
C00767=0.000,-100.950,49.560,0.0000,0.6200,0.7800
C00768=5.040,-100.820,49.550,-0.0300,0.6200,0.7800
C00769=10.040,-100.490,49.560,-0.0200,0.6200,0.7900
C00770=14.930,-100.550,49.940,0.1400,0.5500,0.8200
C00771=17.840,-101.950,50.890,0.2100,0.1700,0.9600
C00772=19.730,-104.630,52.210,0.0600,0.0300,1.0000
C00773=21.340,-108.280,53.580,-0.0300,-0.0100,1.0000
C00774=23.000,-112.380,54.640,-0.0800,-0.0400,1.0000
C00775=25.080,-116.100,55.180,-0.0700,-0.0600,1.0000
C00776=28.920,-118.610,55.460,-0.0200,-0.0500,1.0000
C00777=34.050,-119.490,55.690,0.0000,-0.0300,1.0000
C00778=39.590,-118.480,55.920,0.0000,-0.0000,1.0000
C00779=45.100,-116.570,56.080,0.0000,-0.0000,1.0000
C00780=50.540,-114.320,56.080,0.0000,-0.0000,1.0000
C00781=55.790,-111.770,55.920,0.0000,-0.0000,1.0000
C00782=60.410,-108.570,55.690,0.0200,-0.0200,1.0000
C00783=63.430,-104.320,55.460,0.0500,-0.0200,1.0000
C00784=64.360,-99.830,55.180,0.0900,0.0100,1.0000
C00785=63.200,-95.730,54.640,0.0800,0.0300,1.0000
C00786=61.480,-91.650,53.580,0.0300,0.0100,1.0000
C00787=60.030,-87.930,52.210,-0.0600,-0.0200,1.0000
C00788=59.470,-84.710,50.890,-0.2700,-0.0300,0.9600
C00789=60.540,-81.660,49.940,-0.4900,0.2900,0.8200
C00790=63.960,-78.160,49.560,-0.4200,0.4500,0.7900
C00791=67.730,-74.860,49.550,-0.4100,0.4600,0.7800
C00792=71.380,-71.380,49.560,-0.4400,0.4400,0.7800
C00793=74.860,-67.730,49.550,-0.4600,0.4100,0.7800
C00794=78.160,-63.960,49.560,-0.4500,0.4200,0.7900
C00795=81.660,-60.540,49.940,-0.2900,0.4900,0.8200
C00796=84.710,-59.470,50.890,0.0300,0.2700,0.9600
C00797=87.930,-60.030,52.210,0.0200,0.0600,1.0000
C00798=91.650,-61.480,53.580,-0.0100,-0.0300,1.0000
C00799=95.730,-63.200,54.640,-0.0300,-0.0800,1.0000
C00800=99.830,-64.360,55.180,-0.0100,-0.0900,1.0000
C00801=104.320,-63.430,55.460,0.0200,-0.0500,1.0000
C00802=108.570,-60.410,55.690,0.0200,-0.0200,1.0000
C00803=111.770,-55.790,55.920,0.0000,-0.0000,1.0000
C00804=114.320,-50.540,56.080,0.0000,-0.0000,1.0000
C00805=116.570,-45.100,56.080,0.0000,-0.0000,1.0000
C00806=118.480,-39.590,55.920,0.0000,-0.0000,1.0000
C00807=119.490,-34.050,55.690,0.0300,-0.0000,1.0000
C00808=118.610,-28.920,55.460,0.0500,0.0200,1.0000
C00809=116.100,-25.080,55.180,0.0600,0.0700,1.0000
C00810=112.380,-23.000,54.640,0.0400,0.0800,1.0000
C00811=108.280,-21.340,53.580,0.0100,0.0300,1.0000
C00812=104.630,-19.730,52.210,-0.0300,-0.0600,1.0000
C00813=101.950,-17.840,50.890,-0.1700,-0.2100,0.9600
C00814=100.550,-14.930,49.940,-0.5500,-0.1400,0.8200
C00815=100.490,-10.040,49.560,-0.6200,0.0200,0.7900
C00816=100.820,-5.040,49.550,-0.6200,0.0300,0.7800
C00817=100.950,0.000,49.560,-0.6200,0.0000,0.7800
C00818=100.820,5.040,49.550,-0.6200,-0.0300,0.7800
C00819=100.490,10.040,49.560,-0.6200,-0.0200,0.7900
C00820=100.550,14.930,49.940,-0.5500,0.1400,0.8200
C00821=101.950,17.840,50.890,-0.1700,0.2100,0.9600
C00822=104.630,19.730,52.210,-0.0300,0.0600,1.0000
C00823=108.280,21.340,53.580,0.0100,-0.0300,1.0000
C00824=112.380,23.000,54.640,0.0400,-0.0800,1.0000
C00825=116.100,25.080,55.180,0.0600,-0.0700,1.0000
C00826=118.610,28.920,55.460,0.0500,-0.0200,1.0000
C00827=119.490,34.050,55.690,0.0300,0.0000,1.0000
C00828=118.480,39.590,55.920,0.0000,0.0000,1.0000
C00829=116.570,45.100,56.080,0.0000,0.0000,1.0000
C00830=114.320,50.540,56.080,0.0000,0.0000,1.0000
C00831=111.770,55.790,55.920,0.0000,0.0000,1.0000
C00832=108.570,60.410,55.690,0.0200,0.0200,1.0000
C00833=104.320,63.430,55.460,0.0200,0.0500,1.0000
C00834=99.830,64.360,55.180,-0.0100,0.0900,1.0000
C00835=95.730,63.200,54.640,-0.0300,0.0800,1.0000
C00836=91.650,61.480,53.580,-0.0100,0.0300,1.0000
C00837=87.930,60.030,52.210,0.0200,-0.0600,1.0000
C00838=84.710,59.470,50.890,0.0300,-0.2700,0.9600
C00839=81.660,60.540,49.940,-0.2900,-0.4900,0.8200
C00840=78.160,63.960,49.560,-0.4500,-0.4200,0.7900
C00841=74.860,67.730,49.550,-0.4600,-0.4100,0.7800
C00842=71.380,71.380,49.560,-0.4400,-0.4400,0.7800
C00843=67.730,74.860,49.550,-0.4100,-0.4600,0.7800
C00844=63.960,78.160,49.560,-0.4200,-0.4500,0.7900
C00845=60.540,81.660,49.940,-0.4900,-0.2900,0.8200
C00846=59.470,84.710,50.890,-0.2700,0.0300,0.9600
C00847=60.030,87.930,52.210,-0.0600,0.0200,1.0000
C00848=61.480,91.650,53.580,0.0300,-0.0100,1.0000
C00849=63.200,95.730,54.640,0.0800,-0.0300,1.0000
C00850=64.360,99.830,55.180,0.0900,-0.0100,1.0000
C00851=63.430,104.320,55.460,0.0500,0.0200,1.0000
C00852=60.410,108.570,55.690,0.0200,0.0200,1.0000
C00853=55.790,111.770,55.920,0.0000,0.0000,1.0000
C00854=50.540,114.320,56.080,0.0000,0.0000,1.0000
C00855=45.100,116.570,56.080,0.0000,0.0000,1.0000
C00856=39.590,118.480,55.920,0.0000,0.0000,1.0000
C00857=34.050,119.490,55.690,0.0000,0.0300,1.0000
C00858=28.920,118.610,55.460,-0.0200,0.0500,1.0000
C00859=25.080,116.100,55.180,-0.0700,0.0600,1.0000
C00860=23.000,112.380,54.640,-0.0800,0.0400,1.0000
C00861=21.340,108.280,53.580,-0.0300,0.0100,1.0000
C00862=19.730,104.630,52.210,0.0600,-0.0300,1.0000
C00863=17.840,101.950,50.890,0.2100,-0.1700,0.9600
C00864=14.930,100.550,49.940,0.1400,-0.5500,0.8200
C00865=10.040,100.490,49.560,-0.0200,-0.6200,0.7900
C00866=5.040,100.820,49.550,-0.0300,-0.6200,0.7800
C00867=0.000,100.950,49.560,0.0000,-0.6200,0.7800
C00868=0.000,99.890,50.890,0.0000,-0.6200,0.7800
C00869=4.950,99.770,50.880,-0.0300,-0.6200,0.7800
C00870=9.880,99.450,50.890,-0.0200,-0.6200,0.7800
C00871=14.730,99.540,51.290,0.1500,-0.5400,0.8300
C00872=17.600,101.020,52.290,0.2000,-0.1600,0.9700
C00873=19.440,103.830,53.680,0.0500,-0.0200,1.0000
C00874=21.020,107.660,55.130,-0.0400,0.0200,1.0000
C00875=22.660,111.970,56.260,-0.0900,0.0400,1.0000
C00876=24.700,115.900,56.820,-0.0700,0.0600,1.0000
C00877=28.560,118.570,57.120,-0.0200,0.0500,1.0000
C00878=33.770,119.540,57.360,-0.0000,0.0300,1.0000
C00879=39.410,118.540,57.610,0.0000,0.0000,1.0000
C00880=45.040,116.590,57.780,0.0000,0.0000,1.0000
C00881=50.600,114.290,57.780,0.0000,0.0000,1.0000
C00882=55.960,111.690,57.610,0.0000,0.0000,1.0000
C00883=60.650,108.410,57.360,0.0200,0.0200,1.0000
C00884=63.650,104.040,57.120,0.0500,0.0200,1.0000
C00885=64.480,99.420,56.820,0.1000,-0.0100,1.0000
C00886=63.160,95.200,56.260,0.0900,-0.0400,1.0000
C00887=61.260,90.990,55.130,0.0400,-0.0200,1.0000
C00888=59.670,87.170,53.680,-0.0500,0.0200,1.0000
C00889=58.990,83.880,52.290,-0.2500,0.0300,0.9700
C00890=59.970,80.800,51.290,-0.4900,-0.2800,0.8300
C00891=63.330,77.300,50.890,-0.4200,-0.4500,0.7800
C00892=67.050,74.050,50.880,-0.4200,-0.4600,0.7800
C00893=70.640,70.640,50.890,-0.4400,-0.4400,0.7800
C00894=74.050,67.050,50.880,-0.4600,-0.4200,0.7800
C00895=77.300,63.330,50.890,-0.4500,-0.4200,0.7800
C00896=80.800,59.970,51.290,-0.2800,-0.4900,0.8300
C00897=83.880,58.990,52.290,0.0300,-0.2500,0.9700
C00898=87.170,59.670,53.680,0.0200,-0.0500,1.0000
C00899=90.990,61.260,55.130,-0.0200,0.0400,1.0000
C00900=95.200,63.160,56.260,-0.0400,0.0900,1.0000
C00901=99.420,64.480,56.820,-0.0100,0.1000,1.0000
C00902=104.040,63.650,57.120,0.0200,0.0500,1.0000
C00903=108.410,60.650,57.360,0.0200,0.0200,1.0000
C00904=111.690,55.960,57.610,0.0000,0.0000,1.0000
C00905=114.290,50.600,57.780,0.0000,0.0000,1.0000
C00906=116.590,45.040,57.780,0.0000,0.0000,1.0000
C00907=118.540,39.410,57.610,0.0000,0.0000,1.0000
C00908=119.540,33.770,57.360,0.0300,-0.0000,1.0000
C00909=118.570,28.560,57.120,0.0500,-0.0200,1.0000
C00910=115.900,24.700,56.820,0.0600,-0.0700,1.0000
C00911=111.970,22.660,56.260,0.0400,-0.0900,1.0000
C00912=107.660,21.020,55.130,0.0200,-0.0400,1.0000
C00913=103.830,19.440,53.680,-0.0200,0.0500,1.0000
C00914=101.020,17.600,52.290,-0.1600,0.2000,0.9700
C00915=99.540,14.730,51.290,-0.5400,0.1500,0.8300
C00916=99.450,9.880,50.890,-0.6200,-0.0200,0.7800
C00917=99.770,4.950,50.880,-0.6200,-0.0300,0.7800
C00918=99.890,0.000,50.890,-0.6200,0.0000,0.7800
C00919=99.770,-4.950,50.880,-0.6200,0.0300,0.7800
C00920=99.450,-9.880,50.890,-0.6200,0.0200,0.7800
C00921=99.540,-14.730,51.290,-0.5400,-0.1500,0.8300
C00922=101.020,-17.600,52.290,-0.1600,-0.2000,0.9700
C00923=103.830,-19.440,53.680,-0.0200,-0.0500,1.0000
C00924=107.660,-21.020,55.130,0.0200,0.0400,1.0000
C00925=111.970,-22.660,56.260,0.0400,0.0900,1.0000
C00926=115.900,-24.700,56.820,0.0600,0.0700,1.0000
C00927=118.570,-28.560,57.120,0.0500,0.0200,1.0000
C00928=119.540,-33.770,57.360,0.0300,0.0000,1.0000
C00929=118.540,-39.410,57.610,0.0000,-0.0000,1.0000
C00930=116.590,-45.040,57.780,0.0000,-0.0000,1.0000
C00931=114.290,-50.600,57.780,0.0000,-0.0000,1.0000
C00932=111.690,-55.960,57.610,0.0000,-0.0000,1.0000
C00933=108.410,-60.650,57.360,0.0200,-0.0200,1.0000
C00934=104.040,-63.650,57.120,0.0200,-0.0500,1.0000
C00935=99.420,-64.480,56.820,-0.0100,-0.1000,1.0000
C00936=95.200,-63.160,56.260,-0.0400,-0.0900,1.0000
C00937=90.990,-61.260,55.130,-0.0200,-0.0400,1.0000
C00938=87.170,-59.670,53.680,0.0200,0.0500,1.0000
C00939=83.880,-58.990,52.290,0.0300,0.2500,0.9700
C00940=80.800,-59.970,51.290,-0.2800,0.4900,0.8300
C00941=77.300,-63.330,50.890,-0.4500,0.4200,0.7800
C00942=74.050,-67.050,50.880,-0.4600,0.4200,0.7800
C00943=70.640,-70.640,50.890,-0.4400,0.4400,0.7800
C00944=67.050,-74.050,50.880,-0.4200,0.4600,0.7800
C00945=63.330,-77.300,50.890,-0.4200,0.4500,0.7800
C00946=59.970,-80.800,51.290,-0.4900,0.2800,0.8300
C00947=58.990,-83.880,52.290,-0.2500,-0.0300,0.9700
C00948=59.670,-87.170,53.680,-0.0500,-0.0200,1.0000
C00949=61.260,-90.990,55.130,0.0400,0.0200,1.0000
C00950=63.160,-95.200,56.260,0.0900,0.0400,1.0000
C00951=64.480,-99.420,56.820,0.1000,0.0100,1.0000
C00952=63.650,-104.040,57.120,0.0500,-0.0200,1.0000
C00953=60.650,-108.410,57.360,0.0200,-0.0200,1.0000
C00954=55.960,-111.690,57.610,0.0000,-0.0000,1.0000
C00955=50.600,-114.290,57.780,0.0000,-0.0000,1.0000
C00956=45.040,-116.590,57.780,0.0000,-0.0000,1.0000
C00957=39.410,-118.540,57.610,0.0000,-0.0000,1.0000
C00958=33.770,-119.540,57.360,-0.0000,-0.0300,1.0000
C00959=28.560,-118.570,57.120,-0.0200,-0.0500,1.0000
C00960=24.700,-115.900,56.820,-0.0700,-0.0600,1.0000
C00961=22.660,-111.970,56.260,-0.0900,-0.0400,1.0000
C00962=21.020,-107.660,55.130,-0.0400,-0.0200,1.0000
C00963=19.440,-103.830,53.680,0.0500,0.0200,1.0000
C00964=17.600,-101.020,52.290,0.2000,0.1600,0.9700
C00965=14.730,-99.540,51.290,0.1500,0.5400,0.8300
C00966=9.880,-99.450,50.890,-0.0200,0.6200,0.7800
C00967=4.950,-99.770,50.880,-0.0300,0.6200,0.7800
C00968=0.000,-99.890,50.890,0.0000,0.6200,0.7800
C00969=0.000,-99.890,50.890,0.0000,0.6200,0.7800
C00970=-4.950,-99.770,50.880,0.0300,0.6200,0.7800
C00971=-9.880,-99.450,50.890,0.0200,0.6200,0.7800
C00972=-14.730,-99.540,51.290,-0.1500,0.5400,0.8300
C00973=-17.600,-101.020,52.290,-0.2000,0.1600,0.9700
C00974=-19.440,-103.830,53.680,-0.0500,0.0200,1.0000
C00975=-21.020,-107.660,55.130,0.0400,-0.0200,1.0000
C00976=-22.660,-111.970,56.260,0.0900,-0.0400,1.0000
C00977=-24.700,-115.900,56.820,0.0700,-0.0600,1.0000
C00978=-28.560,-118.570,57.120,0.0200,-0.0500,1.0000
C00979=-33.770,-119.540,57.360,0.0000,-0.0300,1.0000
C00980=-39.410,-118.540,57.610,-0.0000,-0.0000,1.0000
C00981=-45.040,-116.590,57.780,-0.0000,-0.0000,1.0000
C00982=-50.600,-114.290,57.780,-0.0000,-0.0000,1.0000
C00983=-55.960,-111.690,57.610,-0.0000,-0.0000,1.0000
C00984=-60.650,-108.410,57.360,-0.0200,-0.0200,1.0000
C00985=-63.650,-104.040,57.120,-0.0500,-0.0200,1.0000
C00986=-64.480,-99.420,56.820,-0.1000,0.0100,1.0000
C00987=-63.160,-95.200,56.260,-0.0900,0.0400,1.0000
C00988=-61.260,-90.990,55.130,-0.0400,0.0200,1.0000
C00989=-59.670,-87.170,53.680,0.0500,-0.0200,1.0000
C00990=-58.990,-83.880,52.290,0.2500,-0.0300,0.9700
C00991=-59.970,-80.800,51.290,0.4900,0.2800,0.8300
C00992=-63.330,-77.300,50.890,0.4200,0.4500,0.7800
C00993=-67.050,-74.050,50.880,0.4200,0.4600,0.7800
C00994=-70.640,-70.640,50.890,0.4400,0.4400,0.7800
C00995=-74.050,-67.050,50.880,0.4600,0.4200,0.7800
C00996=-77.300,-63.330,50.890,0.4500,0.4200,0.7800
C00997=-80.800,-59.970,51.290,0.2800,0.4900,0.8300
C00998=-83.880,-58.990,52.290,-0.0300,0.2500,0.9700
C00999=-87.170,-59.670,53.680,-0.0200,0.0500,1.0000
C01000=-90.990,-61.260,55.130,0.0200,-0.0400,1.0000
C01001=-95.200,-63.160,56.260,0.0400,-0.0900,1.0000
C01002=-99.420,-64.480,56.820,0.0100,-0.1000,1.0000
C01003=-104.040,-63.650,57.120,-0.0200,-0.0500,1.0000
C01004=-108.410,-60.650,57.360,-0.0200,-0.0200,1.0000
C01005=-111.690,-55.960,57.610,-0.0000,-0.0000,1.0000
C01006=-114.290,-50.600,57.780,-0.0000,-0.0000,1.0000
C01007=-116.590,-45.040,57.780,-0.0000,-0.0000,1.0000
C01008=-118.540,-39.410,57.610,-0.0000,-0.0000,1.0000
C01009=-119.540,-33.770,57.360,-0.0300,0.0000,1.0000
C01010=-118.570,-28.560,57.120,-0.0500,0.0200,1.0000
C01011=-115.900,-24.700,56.820,-0.0600,0.0700,1.0000
C01012=-111.970,-22.660,56.260,-0.0400,0.0900,1.0000
C01013=-107.660,-21.020,55.130,-0.0200,0.0400,1.0000
C01014=-103.830,-19.440,53.680,0.0200,-0.0500,1.0000
C01015=-101.020,-17.600,52.290,0.1600,-0.2000,0.9700
C01016=-99.540,-14.730,51.290,0.5400,-0.1500,0.8300
C01017=-99.450,-9.880,50.890,0.6200,0.0200,0.7800
C01018=-99.770,-4.950,50.880,0.6200,0.0300,0.7800
C01019=-99.890,0.000,50.890,0.6200,-0.0000,0.7800
C01020=-99.770,4.950,50.880,0.6200,-0.0300,0.7800
C01021=-99.450,9.880,50.890,0.6200,-0.0200,0.7800
C01022=-99.540,14.730,51.290,0.5400,0.1500,0.8300
C01023=-101.020,17.600,52.290,0.1600,0.2000,0.9700
C01024=-103.830,19.440,53.680,0.0200,0.0500,1.0000
C01025=-107.660,21.020,55.130,-0.0200,-0.0400,1.0000
C01026=-111.970,22.660,56.260,-0.0400,-0.0900,1.0000
C01027=-115.900,24.700,56.820,-0.0600,-0.0700,1.0000
C01028=-118.570,28.560,57.120,-0.0500,-0.0200,1.0000
C01029=-119.540,33.770,57.360,-0.0300,-0.0000,1.0000
C01030=-118.540,39.410,57.610,-0.0000,0.0000,1.0000
C01031=-116.590,45.040,57.780,-0.0000,0.0000,1.0000
C01032=-114.290,50.600,57.780,-0.0000,0.0000,1.0000
C01033=-111.690,55.960,57.610,-0.0000,0.0000,1.0000
C01034=-108.410,60.650,57.360,-0.0200,0.0200,1.0000
C01035=-104.040,63.650,57.120,-0.0200,0.0500,1.0000
C01036=-99.420,64.480,56.820,0.0100,0.1000,1.0000
C01037=-95.200,63.160,56.260,0.0400,0.0900,1.0000
C01038=-90.990,61.260,55.130,0.0200,0.0400,1.0000
C01039=-87.170,59.670,53.680,-0.0200,-0.0500,1.0000
C01040=-83.880,58.990,52.290,-0.0300,-0.2500,0.9700
C01041=-80.800,59.970,51.290,0.2800,-0.4900,0.8300
C01042=-77.300,63.330,50.890,0.4500,-0.4200,0.7800
C01043=-74.050,67.050,50.880,0.4600,-0.4200,0.7800
C01044=-70.640,70.640,50.890,0.4400,-0.4400,0.7800
C01045=-67.050,74.050,50.880,0.4200,-0.4600,0.7800
C01046=-63.330,77.300,50.890,0.4200,-0.4500,0.7800
C01047=-59.970,80.800,51.290,0.4900,-0.2800,0.8300
C01048=-58.990,83.880,52.290,0.2500,0.0300,0.9700
C01049=-59.670,87.170,53.680,0.0500,0.0200,1.0000
C01050=-61.260,90.990,55.130,-0.0400,-0.0200,1.0000
C01051=-63.160,95.200,56.260,-0.0900,-0.0400,1.0000
C01052=-64.480,99.420,56.820,-0.1000,-0.0100,1.0000
C01053=-63.650,104.040,57.120,-0.0500,0.0200,1.0000
C01054=-60.650,108.410,57.360,-0.0200,0.0200,1.0000
C01055=-55.960,111.690,57.610,-0.0000,0.0000,1.0000
C01056=-50.600,114.290,57.780,-0.0000,0.0000,1.0000
C01057=-45.040,116.590,57.780,-0.0000,0.0000,1.0000
C01058=-39.410,118.540,57.610,-0.0000,0.0000,1.0000
C01059=-33.770,119.540,57.360,0.0000,0.0300,1.0000
C01060=-28.560,118.570,57.120,0.0200,0.0500,1.0000
C01061=-24.700,115.900,56.820,0.0700,0.0600,1.0000
C01062=-22.660,111.970,56.260,0.0900,0.0400,1.0000
C01063=-21.020,107.660,55.130,0.0400,0.0200,1.0000
C01064=-19.440,103.830,53.680,-0.0500,-0.0200,1.0000
C01065=-17.600,101.020,52.290,-0.2000,-0.1600,0.9700
C01066=-14.730,99.540,51.290,-0.1500,-0.5400,0.8300
C01067=-9.880,99.450,50.890,0.0200,-0.6200,0.7800
C01068=-4.950,99.770,50.880,0.0300,-0.6200,0.7800
C01069=0.000,99.890,50.890,0.0000,-0.6200,0.7800
C01070=0.000,98.830,52.220,0.0000,-0.6300,0.7800
C01071=-4.850,98.710,52.200,0.0300,-0.6300,0.7800
C01072=-9.710,98.400,52.220,0.0200,-0.6200,0.7800
C01073=-14.530,98.520,52.640,-0.1600,-0.5400,0.8300
C01074=-17.350,100.090,53.690,-0.1900,-0.1400,0.9700
C01075=-19.160,103.030,55.150,-0.0400,-0.0200,1.0000
C01076=-20.700,107.040,56.680,0.0500,0.0200,1.0000
C01077=-22.310,111.560,57.870,0.0900,0.0400,0.9900
C01078=-24.320,115.690,58.460,0.0800,0.0600,0.9900
C01079=-28.200,118.530,58.780,0.0200,0.0500,1.0000
C01080=-33.480,119.590,59.040,0.0000,0.0300,1.0000
C01081=-39.230,118.600,59.300,-0.0000,0.0000,1.0000
C01082=-44.980,116.620,59.480,-0.0000,0.0000,1.0000
C01083=-50.660,114.260,59.480,-0.0000,0.0000,1.0000
C01084=-56.130,111.600,59.300,-0.0000,0.0000,1.0000
C01085=-60.890,108.240,59.040,-0.0200,0.0200,1.0000
C01086=-63.870,103.750,58.780,-0.0500,0.0200,1.0000
C01087=-64.600,99.000,58.460,-0.1000,-0.0100,0.9900
C01088=-63.110,94.660,57.870,-0.0900,-0.0400,0.9900
C01089=-61.050,90.330,56.680,-0.0500,-0.0200,1.0000
C01090=-59.310,86.400,55.150,0.0400,0.0100,1.0000
C01091=-58.510,83.040,53.690,0.2400,0.0400,0.9700
C01092=-59.390,79.940,52.640,0.5000,-0.2700,0.8300
C01093=-62.710,76.450,52.220,0.4300,-0.4500,0.7800
C01094=-66.370,73.230,52.200,0.4200,-0.4700,0.7800
C01095=-69.880,69.880,52.220,0.4400,-0.4400,0.7800
C01096=-73.230,66.370,52.200,0.4700,-0.4200,0.7800
C01097=-76.440,62.710,52.220,0.4500,-0.4300,0.7800
C01098=-79.940,59.390,52.640,0.2700,-0.5000,0.8300
C01099=-83.040,58.510,53.690,-0.0400,-0.2400,0.9700
C01100=-86.400,59.310,55.150,-0.0100,-0.0400,1.0000
C01101=-90.330,61.050,56.680,0.0200,0.0500,1.0000
C01102=-94.660,63.110,57.870,0.0400,0.0900,0.9900
C01103=-99.000,64.600,58.460,0.0100,0.1000,0.9900
C01104=-103.750,63.870,58.780,-0.0200,0.0500,1.0000
C01105=-108.240,60.890,59.040,-0.0200,0.0200,1.0000
C01106=-111.600,56.130,59.300,-0.0000,0.0000,1.0000
C01107=-114.260,50.660,59.480,-0.0000,0.0000,1.0000
C01108=-116.620,44.980,59.480,-0.0000,0.0000,1.0000
C01109=-118.600,39.230,59.300,-0.0000,0.0000,1.0000
C01110=-119.590,33.480,59.040,-0.0300,-0.0000,1.0000
C01111=-118.530,28.200,58.780,-0.0500,-0.0200,1.0000
C01112=-115.690,24.320,58.460,-0.0600,-0.0800,0.9900
C01113=-111.560,22.310,57.870,-0.0400,-0.0900,0.9900
C01114=-107.040,20.700,56.680,-0.0200,-0.0500,1.0000
C01115=-103.030,19.160,55.150,0.0200,0.0400,1.0000
C01116=-100.090,17.350,53.690,0.1400,0.1900,0.9700
C01117=-98.520,14.530,52.640,0.5400,0.1600,0.8300
C01118=-98.400,9.710,52.220,0.6200,-0.0200,0.7800
C01119=-98.710,4.850,52.200,0.6300,-0.0300,0.7800
C01120=-98.830,0.000,52.220,0.6300,-0.0000,0.7800
C01121=-98.710,-4.850,52.200,0.6300,0.0300,0.7800
C01122=-98.400,-9.710,52.220,0.6200,0.0200,0.7800
C01123=-98.520,-14.530,52.640,0.5400,-0.1600,0.8300
C01124=-100.090,-17.350,53.690,0.1400,-0.1900,0.9700
C01125=-103.030,-19.160,55.150,0.0200,-0.0400,1.0000
C01126=-107.040,-20.700,56.680,-0.0200,0.0500,1.0000
C01127=-111.560,-22.310,57.870,-0.0400,0.0900,0.9900
C01128=-115.690,-24.320,58.460,-0.0600,0.0800,0.9900
C01129=-118.530,-28.200,58.780,-0.0500,0.0200,1.0000
C01130=-119.590,-33.480,59.040,-0.0300,0.0000,1.0000
C01131=-118.600,-39.230,59.300,-0.0000,-0.0000,1.0000
C01132=-116.620,-44.980,59.480,-0.0000,-0.0000,1.0000
C01133=-114.260,-50.660,59.480,-0.0000,-0.0000,1.0000
C01134=-111.600,-56.130,59.300,-0.0000,-0.0000,1.0000
C01135=-108.240,-60.890,59.040,-0.0200,-0.0200,1.0000
C01136=-103.750,-63.870,58.780,-0.0200,-0.0500,1.0000
C01137=-99.000,-64.600,58.460,0.0100,-0.1000,0.9900
C01138=-94.660,-63.110,57.870,0.0400,-0.0900,0.9900
C01139=-90.330,-61.050,56.680,0.0200,-0.0500,1.0000
C01140=-86.400,-59.310,55.150,-0.0100,0.0400,1.0000
C01141=-83.040,-58.510,53.690,-0.0400,0.2400,0.9700
C01142=-79.940,-59.390,52.640,0.2700,0.5000,0.8300
C01143=-76.450,-62.710,52.220,0.4500,0.4300,0.7800
C01144=-73.230,-66.370,52.200,0.4700,0.4200,0.7800
C01145=-69.880,-69.880,52.220,0.4400,0.4400,0.7800
C01146=-66.370,-73.230,52.200,0.4200,0.4700,0.7800
C01147=-62.710,-76.440,52.220,0.4300,0.4500,0.7800
C01148=-59.390,-79.940,52.640,0.5000,0.2700,0.8300
C01149=-58.510,-83.040,53.690,0.2400,-0.0400,0.9700
C01150=-59.310,-86.400,55.150,0.0400,-0.0100,1.0000
C01151=-61.050,-90.330,56.680,-0.0500,0.0200,1.0000
C01152=-63.110,-94.660,57.870,-0.0900,0.0400,0.9900
C01153=-64.600,-99.000,58.460,-0.1000,0.0100,0.9900
C01154=-63.870,-103.750,58.780,-0.0500,-0.0200,1.0000
C01155=-60.890,-108.240,59.040,-0.0200,-0.0200,1.0000
C01156=-56.130,-111.600,59.300,-0.0000,-0.0000,1.0000
C01157=-50.660,-114.260,59.480,-0.0000,-0.0000,1.0000
C01158=-44.980,-116.620,59.480,-0.0000,-0.0000,1.0000
C01159=-39.230,-118.600,59.300,-0.0000,-0.0000,1.0000
C01160=-33.480,-119.590,59.040,0.0000,-0.0300,1.0000
C01161=-28.200,-118.530,58.780,0.0200,-0.0500,1.0000
C01162=-24.320,-115.690,58.460,0.0800,-0.0600,0.9900
C01163=-22.310,-111.560,57.870,0.0900,-0.0400,0.9900
C01164=-20.700,-107.040,56.680,0.0500,-0.0200,1.0000
C01165=-19.160,-103.030,55.150,-0.0400,0.0200,1.0000
C01166=-17.350,-100.090,53.690,-0.1900,0.1400,0.9700
C01167=-14.530,-98.520,52.640,-0.1600,0.5400,0.8300
C01168=-9.710,-98.400,52.220,0.0200,0.6200,0.7800
C01169=-4.850,-98.710,52.200,0.0300,0.6300,0.7800
C01170=0.000,-98.830,52.220,0.0000,0.6300,0.7800
C01171=0.000,-98.830,52.220,0.0000,0.6300,0.7800
C01172=4.850,-98.710,52.200,-0.0300,0.6300,0.7800
C01173=9.710,-98.400,52.220,-0.0200,0.6200,0.7800
C01174=14.530,-98.520,52.640,0.1600,0.5400,0.8300
C01175=17.350,-100.090,53.690,0.1900,0.1400,0.9700
C01176=19.160,-103.030,55.150,0.0400,0.0200,1.0000
C01177=20.700,-107.040,56.680,-0.0500,-0.0200,1.0000
C01178=22.310,-111.560,57.870,-0.0900,-0.0400,0.9900
C01179=24.320,-115.690,58.460,-0.0800,-0.0600,0.9900
C01180=28.200,-118.530,58.780,-0.0200,-0.0500,1.0000
C01181=33.480,-119.590,59.040,-0.0000,-0.0300,1.0000
C01182=39.230,-118.600,59.300,0.0000,-0.0000,1.0000
C01183=44.980,-116.620,59.480,0.0000,-0.0000,1.0000
C01184=50.660,-114.260,59.480,0.0000,-0.0000,1.0000
C01185=56.130,-111.600,59.300,0.0000,-0.0000,1.0000
C01186=60.890,-108.240,59.040,0.0200,-0.0200,1.0000
C01187=63.870,-103.750,58.780,0.0500,-0.0200,1.0000
C01188=64.600,-99.000,58.460,0.1000,0.0100,0.9900
C01189=63.110,-94.660,57.870,0.0900,0.0400,0.9900
C01190=61.050,-90.330,56.680,0.0500,0.0200,1.0000
C01191=59.310,-86.400,55.150,-0.0400,-0.0100,1.0000
C01192=58.510,-83.040,53.690,-0.2400,-0.0400,0.9700
C01193=59.390,-79.940,52.640,-0.5000,0.2700,0.8300
C01194=62.710,-76.450,52.220,-0.4300,0.4500,0.7800
C01195=66.370,-73.230,52.200,-0.4200,0.4700,0.7800
C01196=69.880,-69.880,52.220,-0.4400,0.4400,0.7800
C01197=73.230,-66.370,52.200,-0.4700,0.4200,0.7800
C01198=76.440,-62.710,52.220,-0.4500,0.4300,0.7800
C01199=79.940,-59.390,52.640,-0.2700,0.5000,0.8300
C01200=83.040,-58.510,53.690,0.0400,0.2400,0.9700
C01201=86.400,-59.310,55.150,0.0100,0.0400,1.0000
C01202=90.330,-61.050,56.680,-0.0200,-0.0500,1.0000
C01203=94.660,-63.110,57.870,-0.0400,-0.0900,0.9900
C01204=99.000,-64.600,58.460,-0.0100,-0.1000,0.9900
C01205=103.750,-63.870,58.780,0.0200,-0.0500,1.0000
C01206=108.240,-60.890,59.040,0.0200,-0.0200,1.0000
C01207=111.600,-56.130,59.300,0.0000,-0.0000,1.0000
C01208=114.260,-50.660,59.480,0.0000,-0.0000,1.0000
C01209=116.620,-44.980,59.480,0.0000,-0.0000,1.0000
C01210=118.600,-39.230,59.300,0.0000,-0.0000,1.0000
C01211=119.590,-33.480,59.040,0.0300,0.0000,1.0000
C01212=118.530,-28.200,58.780,0.0500,0.0200,1.0000
C01213=115.690,-24.320,58.460,0.0600,0.0800,0.9900
C01214=111.560,-22.310,57.870,0.0400,0.0900,0.9900
C01215=107.040,-20.700,56.680,0.0200,0.0500,1.0000
C01216=103.030,-19.160,55.150,-0.0200,-0.0400,1.0000
C01217=100.090,-17.350,53.690,-0.1400,-0.1900,0.9700
C01218=98.520,-14.530,52.640,-0.5400,-0.1600,0.8300
C01219=98.400,-9.710,52.220,-0.6200,0.0200,0.7800
C01220=98.710,-4.850,52.200,-0.6300,0.0300,0.7800
C01221=98.830,0.000,52.220,-0.6300,0.0000,0.7800
C01222=98.710,4.850,52.200,-0.6300,-0.0300,0.7800
C01223=98.400,9.710,52.220,-0.6200,-0.0200,0.7800
C01224=98.520,14.530,52.640,-0.5400,0.1600,0.8300
C01225=100.090,17.350,53.690,-0.1400,0.1900,0.9700
C01226=103.030,19.160,55.150,-0.0200,0.0400,1.0000
C01227=107.040,20.700,56.680,0.0200,-0.0500,1.0000
C01228=111.560,22.310,57.870,0.0400,-0.0900,0.9900
C01229=115.690,24.320,58.460,0.0600,-0.0800,0.9900
C01230=118.530,28.200,58.780,0.0500,-0.0200,1.0000
C01231=119.590,33.480,59.040,0.0300,-0.0000,1.0000
C01232=118.600,39.230,59.300,0.0000,0.0000,1.0000
C01233=116.620,44.980,59.480,0.0000,0.0000,1.0000
C01234=114.260,50.660,59.480,0.0000,0.0000,1.0000
C01235=111.600,56.130,59.300,0.0000,0.0000,1.0000
C01236=108.240,60.890,59.040,0.0200,0.0200,1.0000
C01237=103.750,63.870,58.780,0.0200,0.0500,1.0000
C01238=99.000,64.600,58.460,-0.0100,0.1000,0.9900
C01239=94.660,63.110,57.870,-0.0400,0.0900,0.9900
C01240=90.330,61.050,56.680,-0.0200,0.0500,1.0000
C01241=86.400,59.310,55.150,0.0100,-0.0400,1.0000
C01242=83.040,58.510,53.690,0.0400,-0.2400,0.9700
C01243=79.940,59.390,52.640,-0.2700,-0.5000,0.8300
C01244=76.450,62.710,52.220,-0.4500,-0.4300,0.7800
C01245=73.230,66.370,52.200,-0.4700,-0.4200,0.7800
C01246=69.880,69.880,52.220,-0.4400,-0.4400,0.7800
C01247=66.370,73.230,52.200,-0.4200,-0.4700,0.7800
C01248=62.710,76.440,52.220,-0.4300,-0.4500,0.7800
C01249=59.390,79.940,52.640,-0.5000,-0.2700,0.8300
C01250=58.510,83.040,53.690,-0.2400,0.0400,0.9700
C01251=59.310,86.400,55.150,-0.0400,0.0100,1.0000
C01252=61.050,90.330,56.680,0.0500,-0.0200,1.0000
C01253=63.110,94.660,57.870,0.0900,-0.0400,0.9900
C01254=64.600,99.000,58.460,0.1000,-0.0100,0.9900
C01255=63.870,103.750,58.780,0.0500,0.0200,1.0000
C01256=60.890,108.240,59.040,0.0200,0.0200,1.0000
C01257=56.130,111.600,59.300,0.0000,0.0000,1.0000
C01258=50.660,114.260,59.480,0.0000,0.0000,1.0000
C01259=44.980,116.620,59.480,0.0000,0.0000,1.0000
C01260=39.230,118.600,59.300,0.0000,0.0000,1.0000
C01261=33.480,119.590,59.040,-0.0000,0.0300,1.0000
C01262=28.200,118.530,58.780,-0.0200,0.0500,1.0000
C01263=24.320,115.690,58.460,-0.0800,0.0600,0.9900
C01264=22.310,111.560,57.870,-0.0900,0.0400,0.9900
C01265=20.700,107.040,56.680,-0.0500,0.0200,1.0000
C01266=19.160,103.030,55.150,0.0400,-0.0200,1.0000
C01267=17.350,100.090,53.690,0.1900,-0.1400,0.9700
C01268=14.530,98.520,52.640,0.1600,-0.5400,0.8300
C01269=9.710,98.400,52.220,-0.0200,-0.6200,0.7800
C01270=4.850,98.710,52.200,-0.0300,-0.6300,0.7800
C01271=0.000,98.830,52.220,0.0000,-0.6300,0.7800
C01272=0.000,97.760,53.540,0.0000,-0.6300,0.7800
C01273=4.750,97.650,53.530,-0.0300,-0.6300,0.7800
C01274=9.550,97.340,53.550,-0.0200,-0.6300,0.7800
C01275=14.330,97.500,53.980,0.1700,-0.5300,0.8300
C01276=17.100,99.150,55.090,0.1800,-0.1200,0.9800
C01277=18.870,102.230,56.620,0.0300,-0.0100,1.0000
C01278=20.390,106.420,58.230,-0.0600,0.0200,1.0000
C01279=21.970,111.150,59.480,-0.1000,0.0400,0.9900
C01280=23.950,115.480,60.110,-0.0900,0.0700,0.9900
C01281=27.840,118.480,60.440,-0.0300,0.0600,1.0000
C01282=33.200,119.650,60.710,-0.0000,0.0300,1.0000
C01283=39.050,118.660,60.990,0.0000,0.0000,1.0000
C01284=44.910,116.640,61.180,0.0000,0.0000,1.0000
C01285=50.720,114.240,61.180,0.0000,0.0000,1.0000
C01286=56.300,111.510,60.990,0.0000,0.0000,1.0000
C01287=61.130,108.080,60.710,0.0300,0.0200,1.0000
C01288=64.090,103.470,60.440,0.0600,0.0200,1.0000
C01289=64.730,98.590,60.110,0.1100,-0.0200,0.9900
C01290=63.060,94.130,59.480,0.1000,-0.0400,0.9900
C01291=60.830,89.660,58.230,0.0600,-0.0300,1.0000
C01292=58.940,85.630,56.620,-0.0300,0.0100,1.0000
C01293=58.020,82.200,55.090,-0.2200,0.0400,0.9800
C01294=58.810,79.080,53.980,-0.5000,-0.2500,0.8300
C01295=62.080,75.580,53.550,-0.4300,-0.4500,0.7800
C01296=65.690,72.410,53.530,-0.4200,-0.4700,0.7800
C01297=69.130,69.130,53.540,-0.4400,-0.4400,0.7800
C01298=72.410,65.690,53.530,-0.4700,-0.4200,0.7800
C01299=75.580,62.080,53.550,-0.4500,-0.4300,0.7800
C01300=79.080,58.810,53.980,-0.2500,-0.5000,0.8300
C01301=82.200,58.020,55.090,0.0400,-0.2200,0.9800
C01302=85.630,58.940,56.620,0.0100,-0.0300,1.0000
C01303=89.660,60.830,58.230,-0.0300,0.0600,1.0000
C01304=94.130,63.060,59.480,-0.0400,0.1000,0.9900
C01305=98.590,64.730,60.110,-0.0200,0.1100,0.9900
C01306=103.470,64.090,60.440,0.0200,0.0600,1.0000
C01307=108.080,61.130,60.710,0.0200,0.0300,1.0000
C01308=111.510,56.300,60.990,0.0000,0.0000,1.0000
C01309=114.240,50.720,61.180,0.0000,0.0000,1.0000
C01310=116.640,44.910,61.180,0.0000,0.0000,1.0000
C01311=118.660,39.050,60.990,0.0000,0.0000,1.0000
C01312=119.650,33.200,60.710,0.0300,-0.0000,1.0000
C01313=118.480,27.840,60.440,0.0600,-0.0300,1.0000
C01314=115.480,23.950,60.110,0.0700,-0.0900,0.9900
C01315=111.150,21.970,59.480,0.0400,-0.1000,0.9900
C01316=106.420,20.390,58.230,0.0200,-0.0600,1.0000
C01317=102.230,18.870,56.620,-0.0100,0.0300,1.0000
C01318=99.150,17.100,55.090,-0.1200,0.1800,0.9800
C01319=97.500,14.330,53.980,-0.5300,0.1700,0.8300
C01320=97.340,9.550,53.550,-0.6300,-0.0200,0.7800
C01321=97.650,4.750,53.530,-0.6300,-0.0300,0.7800
C01322=97.760,0.000,53.540,-0.6300,0.0000,0.7800
C01323=97.650,-4.750,53.530,-0.6300,0.0300,0.7800
C01324=97.340,-9.550,53.550,-0.6300,0.0200,0.7800
C01325=97.500,-14.330,53.980,-0.5300,-0.1700,0.8300
C01326=99.150,-17.100,55.090,-0.1200,-0.1800,0.9800
C01327=102.230,-18.870,56.620,-0.0100,-0.0300,1.0000
C01328=106.420,-20.390,58.230,0.0200,0.0600,1.0000
C01329=111.150,-21.970,59.480,0.0400,0.1000,0.9900
C01330=115.480,-23.950,60.110,0.0700,0.0900,0.9900
C01331=118.480,-27.840,60.440,0.0600,0.0300,1.0000
C01332=119.650,-33.200,60.710,0.0300,0.0000,1.0000
C01333=118.660,-39.050,60.990,0.0000,-0.0000,1.0000
C01334=116.640,-44.910,61.180,0.0000,-0.0000,1.0000
C01335=114.240,-50.720,61.180,0.0000,-0.0000,1.0000
C01336=111.510,-56.300,60.990,0.0000,-0.0000,1.0000
C01337=108.080,-61.130,60.710,0.0200,-0.0300,1.0000
C01338=103.470,-64.090,60.440,0.0200,-0.0600,1.0000
C01339=98.590,-64.730,60.110,-0.0200,-0.1100,0.9900
C01340=94.130,-63.060,59.480,-0.0400,-0.1000,0.9900
C01341=89.660,-60.830,58.230,-0.0300,-0.0600,1.0000
C01342=85.630,-58.940,56.620,0.0100,0.0300,1.0000
C01343=82.200,-58.020,55.090,0.0400,0.2200,0.9800
C01344=79.080,-58.810,53.980,-0.2500,0.5000,0.8300
C01345=75.580,-62.080,53.550,-0.4500,0.4300,0.7800
C01346=72.410,-65.690,53.530,-0.4700,0.4200,0.7800
C01347=69.130,-69.130,53.540,-0.4400,0.4400,0.7800
C01348=65.690,-72.410,53.530,-0.4200,0.4700,0.7800
C01349=62.080,-75.580,53.550,-0.4300,0.4500,0.7800
C01350=58.810,-79.080,53.980,-0.5000,0.2500,0.8300
C01351=58.020,-82.200,55.090,-0.2200,-0.0400,0.9800
C01352=58.940,-85.630,56.620,-0.0300,-0.0100,1.0000
C01353=60.830,-89.660,58.230,0.0600,0.0300,1.0000
C01354=63.060,-94.130,59.480,0.1000,0.0400,0.9900
C01355=64.730,-98.590,60.110,0.1100,0.0200,0.9900
C01356=64.090,-103.470,60.440,0.0600,-0.0200,1.0000
C01357=61.130,-108.080,60.710,0.0300,-0.0200,1.0000
C01358=56.300,-111.510,60.990,0.0000,-0.0000,1.0000
C01359=50.720,-114.240,61.180,0.0000,-0.0000,1.0000
C01360=44.910,-116.640,61.180,0.0000,-0.0000,1.0000
C01361=39.050,-118.660,60.990,0.0000,-0.0000,1.0000
C01362=33.200,-119.650,60.710,-0.0000,-0.0300,1.0000
C01363=27.840,-118.480,60.440,-0.0300,-0.0600,1.0000
C01364=23.950,-115.480,60.110,-0.0900,-0.0700,0.9900
C01365=21.970,-111.150,59.480,-0.1000,-0.0400,0.9900
C01366=20.390,-106.420,58.230,-0.0600,-0.0200,1.0000
C01367=18.870,-102.230,56.620,0.0300,0.0100,1.0000
C01368=17.100,-99.150,55.090,0.1800,0.1200,0.9800
C01369=14.330,-97.500,53.980,0.1700,0.5300,0.8300
C01370=9.550,-97.340,53.550,-0.0200,0.6300,0.7800
C01371=4.750,-97.650,53.530,-0.0300,0.6300,0.7800
C01372=0.000,-97.760,53.540,0.0000,0.6300,0.7800
C01373=0.000,-97.760,53.540,0.0000,0.6300,0.7800
C01374=-4.750,-97.650,53.530,0.0300,0.6300,0.7800
C01375=-9.550,-97.340,53.550,0.0200,0.6300,0.7800
C01376=-14.330,-97.500,53.980,-0.1700,0.5300,0.8300
C01377=-17.100,-99.150,55.090,-0.1800,0.1200,0.9800
C01378=-18.870,-102.230,56.620,-0.0300,0.0100,1.0000
C01379=-20.390,-106.420,58.230,0.0600,-0.0200,1.0000
C01380=-21.970,-111.150,59.480,0.1000,-0.0400,0.9900
C01381=-23.950,-115.480,60.110,0.0900,-0.0700,0.9900
C01382=-27.840,-118.480,60.440,0.0300,-0.0600,1.0000
C01383=-33.200,-119.650,60.710,0.0000,-0.0300,1.0000
C01384=-39.050,-118.660,60.990,-0.0000,-0.0000,1.0000
C01385=-44.910,-116.640,61.180,-0.0000,-0.0000,1.0000
C01386=-50.720,-114.240,61.180,-0.0000,-0.0000,1.0000
C01387=-56.300,-111.510,60.990,-0.0000,-0.0000,1.0000
C01388=-61.130,-108.080,60.710,-0.0300,-0.0200,1.0000
C01389=-64.090,-103.470,60.440,-0.0600,-0.0200,1.0000
C01390=-64.730,-98.590,60.110,-0.1100,0.0200,0.9900
C01391=-63.060,-94.130,59.480,-0.1000,0.0400,0.9900
C01392=-60.830,-89.660,58.230,-0.0600,0.0300,1.0000
C01393=-58.940,-85.630,56.620,0.0300,-0.0100,1.0000
C01394=-58.020,-82.200,55.090,0.2200,-0.0400,0.9800
C01395=-58.810,-79.080,53.980,0.5000,0.2500,0.8300
C01396=-62.080,-75.580,53.550,0.4300,0.4500,0.7800
C01397=-65.690,-72.410,53.530,0.4200,0.4700,0.7800
C01398=-69.130,-69.130,53.540,0.4400,0.4400,0.7800
C01399=-72.410,-65.690,53.530,0.4700,0.4200,0.7800
C01400=-75.580,-62.080,53.550,0.4500,0.4300,0.7800
C01401=-79.080,-58.810,53.980,0.2500,0.5000,0.8300
C01402=-82.200,-58.020,55.090,-0.0400,0.2200,0.9800
C01403=-85.630,-58.940,56.620,-0.0100,0.0300,1.0000
C01404=-89.660,-60.830,58.230,0.0300,-0.0600,1.0000
C01405=-94.130,-63.060,59.480,0.0400,-0.1000,0.9900
C01406=-98.590,-64.730,60.110,0.0200,-0.1100,0.9900
C01407=-103.470,-64.090,60.440,-0.0200,-0.0600,1.0000
C01408=-108.080,-61.130,60.710,-0.0200,-0.0300,1.0000
C01409=-111.510,-56.300,60.990,-0.0000,-0.0000,1.0000
C01410=-114.240,-50.720,61.180,-0.0000,-0.0000,1.0000
C01411=-116.640,-44.910,61.180,-0.0000,-0.0000,1.0000
C01412=-118.660,-39.050,60.990,-0.0000,-0.0000,1.0000
C01413=-119.650,-33.200,60.710,-0.0300,0.0000,1.0000
C01414=-118.480,-27.840,60.440,-0.0600,0.0300,1.0000
C01415=-115.480,-23.950,60.110,-0.0700,0.0900,0.9900
C01416=-111.150,-21.970,59.480,-0.0400,0.1000,0.9900
C01417=-106.420,-20.390,58.230,-0.0200,0.0600,1.0000
C01418=-102.230,-18.870,56.620,0.0100,-0.0300,1.0000
C01419=-99.150,-17.100,55.090,0.1200,-0.1800,0.9800
C01420=-97.500,-14.330,53.980,0.5300,-0.1700,0.8300
C01421=-97.340,-9.550,53.550,0.6300,0.0200,0.7800
C01422=-97.650,-4.750,53.530,0.6300,0.0300,0.7800
C01423=-97.760,0.000,53.540,0.6300,-0.0000,0.7800
C01424=-97.650,4.750,53.530,0.6300,-0.0300,0.7800
C01425=-97.340,9.550,53.550,0.6300,-0.0200,0.7800
C01426=-97.500,14.330,53.980,0.5300,0.1700,0.8300
C01427=-99.150,17.100,55.090,0.1200,0.1800,0.9800
C01428=-102.230,18.870,56.620,0.0100,0.0300,1.0000
C01429=-106.420,20.390,58.230,-0.0200,-0.0600,1.0000
C01430=-111.150,21.970,59.480,-0.0400,-0.1000,0.9900
C01431=-115.480,23.950,60.110,-0.0700,-0.0900,0.9900
C01432=-118.480,27.840,60.440,-0.0600,-0.0300,1.0000
C01433=-119.650,33.200,60.710,-0.0300,-0.0000,1.0000
C01434=-118.660,39.050,60.990,-0.0000,0.0000,1.0000
C01435=-116.640,44.910,61.180,-0.0000,0.0000,1.0000
C01436=-114.240,50.720,61.180,-0.0000,0.0000,1.0000
C01437=-111.510,56.300,60.990,-0.0000,0.0000,1.0000
C01438=-108.080,61.130,60.710,-0.0200,0.0300,1.0000
C01439=-103.470,64.090,60.440,-0.0200,0.0600,1.0000
C01440=-98.590,64.730,60.110,0.0200,0.1100,0.9900
C01441=-94.130,63.060,59.480,0.0400,0.1000,0.9900
C01442=-89.660,60.830,58.230,0.0300,0.0600,1.0000
C01443=-85.630,58.940,56.620,-0.0100,-0.0300,1.0000
C01444=-82.200,58.020,55.090,-0.0400,-0.2200,0.9800
C01445=-79.080,58.810,53.980,0.2500,-0.5000,0.8300
C01446=-75.580,62.080,53.550,0.4500,-0.4300,0.7800
C01447=-72.410,65.690,53.530,0.4700,-0.4200,0.7800
C01448=-69.130,69.130,53.540,0.4400,-0.4400,0.7800
C01449=-65.690,72.410,53.530,0.4200,-0.4700,0.7800
C01450=-62.080,75.580,53.550,0.4300,-0.4500,0.7800
C01451=-58.810,79.080,53.980,0.5000,-0.2500,0.8300
C01452=-58.020,82.200,55.090,0.2200,0.0400,0.9800
C01453=-58.940,85.630,56.620,0.0300,0.0100,1.0000
C01454=-60.830,89.660,58.230,-0.0600,-0.0300,1.0000
C01455=-63.060,94.130,59.480,-0.1000,-0.0400,0.9900
C01456=-64.730,98.590,60.110,-0.1100,-0.0200,0.9900
C01457=-64.090,103.470,60.440,-0.0600,0.0200,1.0000
C01458=-61.130,108.080,60.710,-0.0300,0.0200,1.0000
C01459=-56.300,111.510,60.990,-0.0000,0.0000,1.0000
C01460=-50.720,114.240,61.180,-0.0000,0.0000,1.0000
C01461=-44.910,116.640,61.180,-0.0000,0.0000,1.0000
C01462=-39.050,118.660,60.990,-0.0000,0.0000,1.0000
C01463=-33.200,119.650,60.710,0.0000,0.0300,1.0000
C01464=-27.840,118.480,60.440,0.0300,0.0600,1.0000
C01465=-23.950,115.480,60.110,0.0900,0.0700,0.9900
C01466=-21.970,111.150,59.480,0.1000,0.0400,0.9900
C01467=-20.390,106.420,58.230,0.0600,0.0200,1.0000
C01468=-18.870,102.230,56.620,-0.0300,-0.0100,1.0000
C01469=-17.100,99.150,55.090,-0.1800,-0.1200,0.9800
C01470=-14.330,97.500,53.980,-0.1700,-0.5300,0.8300
C01471=-9.550,97.340,53.550,0.0200,-0.6300,0.7800
C01472=-4.750,97.650,53.530,0.0300,-0.6300,0.7800
C01473=0.000,97.760,53.540,0.0000,-0.6300,0.7800
C01474=0.000,96.690,54.860,0.0000,-0.6300,0.7800
C01475=-4.650,96.580,54.850,0.0300,-0.6300,0.7800
C01476=-9.390,96.280,54.870,0.0100,-0.6300,0.7800
C01477=-14.130,96.480,55.320,-0.1800,-0.5300,0.8300
C01478=-16.850,98.210,56.480,-0.1700,-0.1100,0.9800
C01479=-18.580,101.420,58.090,-0.0200,-0.0100,1.0000
C01480=-20.070,105.790,59.780,0.0700,0.0200,1.0000
C01481=-21.620,110.740,61.090,0.1100,0.0400,0.9900
C01482=-23.570,115.280,61.750,0.0900,0.0700,0.9900
C01483=-27.490,118.440,62.100,0.0300,0.0600,1.0000
C01484=-32.920,119.700,62.390,0.0000,0.0400,1.0000
C01485=-38.860,118.720,62.680,-0.0000,0.0000,1.0000
C01486=-44.850,116.670,62.870,-0.0000,0.0000,1.0000
C01487=-50.780,114.210,62.870,-0.0000,0.0000,1.0000
C01488=-56.470,111.430,62.680,-0.0000,0.0000,1.0000
C01489=-61.360,107.910,62.390,-0.0300,0.0200,1.0000
C01490=-64.320,103.190,62.100,-0.0600,0.0200,1.0000
C01491=-64.850,98.180,61.750,-0.1100,-0.0200,0.9900
C01492=-63.020,93.590,61.090,-0.1000,-0.0500,0.9900
C01493=-60.620,89.000,59.780,-0.0600,-0.0300,1.0000
C01494=-58.580,84.850,58.090,0.0200,0.0100,1.0000
C01495=-57.530,81.360,56.480,0.2000,0.0500,0.9800
C01496=-58.230,78.210,55.320,0.5000,-0.2400,0.8300
C01497=-61.450,74.720,54.870,0.4300,-0.4500,0.7800
C01498=-65.000,71.580,54.850,0.4200,-0.4700,0.7800
C01499=-68.370,68.370,54.860,0.4500,-0.4500,0.7800
C01500=-71.580,65.000,54.850,0.4700,-0.4200,0.7800
C01501=-74.720,61.450,54.870,0.4500,-0.4300,0.7800
C01502=-78.210,58.230,55.320,0.2400,-0.5000,0.8300
C01503=-81.360,57.530,56.480,-0.0500,-0.2000,0.9800
C01504=-84.850,58.580,58.090,-0.0100,-0.0200,1.0000
C01505=-89.000,60.620,59.780,0.0300,0.0600,1.0000
C01506=-93.590,63.020,61.090,0.0500,0.1000,0.9900
C01507=-98.180,64.850,61.750,0.0200,0.1100,0.9900
C01508=-103.190,64.320,62.100,-0.0200,0.0600,1.0000
C01509=-107.910,61.360,62.390,-0.0200,0.0300,1.0000
C01510=-111.430,56.470,62.680,-0.0000,0.0000,1.0000
C01511=-114.210,50.780,62.870,-0.0000,0.0000,1.0000
C01512=-116.670,44.850,62.870,-0.0000,0.0000,1.0000
C01513=-118.720,38.860,62.680,-0.0000,0.0000,1.0000
C01514=-119.700,32.920,62.390,-0.0400,-0.0000,1.0000
C01515=-118.440,27.490,62.100,-0.0600,-0.0300,1.0000
C01516=-115.280,23.570,61.750,-0.0700,-0.0900,0.9900
C01517=-110.740,21.620,61.090,-0.0400,-0.1100,0.9900
C01518=-105.790,20.070,59.780,-0.0200,-0.0700,1.0000
C01519=-101.420,18.580,58.090,0.0100,0.0200,1.0000
C01520=-98.210,16.850,56.480,0.1100,0.1700,0.9800
C01521=-96.480,14.130,55.320,0.5300,0.1800,0.8300
C01522=-96.280,9.390,54.870,0.6300,-0.0100,0.7800
C01523=-96.580,4.650,54.850,0.6300,-0.0300,0.7800
C01524=-96.690,0.000,54.860,0.6300,-0.0000,0.7800
C01525=-96.580,-4.650,54.850,0.6300,0.0300,0.7800
C01526=-96.280,-9.390,54.870,0.6300,0.0100,0.7800
C01527=-96.480,-14.130,55.320,0.5300,-0.1800,0.8300
C01528=-98.210,-16.850,56.480,0.1100,-0.1700,0.9800
C01529=-101.420,-18.580,58.090,0.0100,-0.0200,1.0000
C01530=-105.790,-20.070,59.780,-0.0200,0.0700,1.0000
C01531=-110.740,-21.620,61.090,-0.0400,0.1100,0.9900
C01532=-115.280,-23.570,61.750,-0.0700,0.0900,0.9900
C01533=-118.440,-27.490,62.100,-0.0600,0.0300,1.0000
C01534=-119.700,-32.920,62.390,-0.0400,0.0000,1.0000
C01535=-118.720,-38.860,62.680,-0.0000,-0.0000,1.0000
C01536=-116.670,-44.850,62.870,-0.0000,-0.0000,1.0000
C01537=-114.210,-50.780,62.870,-0.0000,-0.0000,1.0000
C01538=-111.430,-56.470,62.680,-0.0000,-0.0000,1.0000
C01539=-107.910,-61.360,62.390,-0.0200,-0.0300,1.0000
C01540=-103.190,-64.320,62.100,-0.0200,-0.0600,1.0000
C01541=-98.180,-64.850,61.750,0.0200,-0.1100,0.9900
C01542=-93.590,-63.020,61.090,0.0500,-0.1000,0.9900
C01543=-89.000,-60.620,59.780,0.0300,-0.0600,1.0000
C01544=-84.850,-58.580,58.090,-0.0100,0.0200,1.0000
C01545=-81.360,-57.530,56.480,-0.0500,0.2000,0.9800
C01546=-78.210,-58.230,55.320,0.2400,0.5000,0.8300
C01547=-74.720,-61.450,54.870,0.4500,0.4300,0.7800
C01548=-71.580,-65.000,54.850,0.4700,0.4200,0.7800
C01549=-68.370,-68.370,54.860,0.4500,0.4500,0.7800
C01550=-65.000,-71.580,54.850,0.4200,0.4700,0.7800
C01551=-61.450,-74.720,54.870,0.4300,0.4500,0.7800
C01552=-58.230,-78.210,55.320,0.5000,0.2400,0.8300
C01553=-57.530,-81.360,56.480,0.2000,-0.0500,0.9800
C01554=-58.580,-84.850,58.090,0.0200,-0.0100,1.0000
C01555=-60.620,-89.000,59.780,-0.0600,0.0300,1.0000
C01556=-63.020,-93.590,61.090,-0.1000,0.0500,0.9900
C01557=-64.850,-98.180,61.750,-0.1100,0.0200,0.9900
C01558=-64.320,-103.190,62.100,-0.0600,-0.0200,1.0000
C01559=-61.360,-107.910,62.390,-0.0300,-0.0200,1.0000
C01560=-56.470,-111.430,62.680,-0.0000,-0.0000,1.0000
C01561=-50.780,-114.210,62.870,-0.0000,-0.0000,1.0000
C01562=-44.850,-116.670,62.870,-0.0000,-0.0000,1.0000
C01563=-38.860,-118.720,62.680,-0.0000,-0.0000,1.0000
C01564=-32.920,-119.700,62.390,0.0000,-0.0400,1.0000
C01565=-27.490,-118.440,62.100,0.0300,-0.0600,1.0000
C01566=-23.570,-115.280,61.750,0.0900,-0.0700,0.9900
C01567=-21.620,-110.740,61.090,0.1100,-0.0400,0.9900
C01568=-20.070,-105.790,59.780,0.0700,-0.0200,1.0000
C01569=-18.580,-101.420,58.090,-0.0200,0.0100,1.0000
C01570=-16.850,-98.210,56.480,-0.1700,0.1100,0.9800
C01571=-14.130,-96.480,55.320,-0.1800,0.5300,0.8300
C01572=-9.390,-96.280,54.870,0.0100,0.6300,0.7800
C01573=-4.650,-96.580,54.850,0.0300,0.6300,0.7800
C01574=0.000,-96.690,54.860,0.0000,0.6300,0.7800
C01575=0.000,-96.690,54.860,0.0000,0.6300,0.7800
C01576=4.650,-96.580,54.850,-0.0300,0.6300,0.7800
C01577=9.390,-96.280,54.870,-0.0100,0.6300,0.7800
C01578=14.130,-96.480,55.320,0.1800,0.5300,0.8300
C01579=16.850,-98.210,56.480,0.1700,0.1100,0.9800
C01580=18.580,-101.420,58.090,0.0200,0.0100,1.0000
C01581=20.070,-105.790,59.780,-0.0700,-0.0200,1.0000
C01582=21.620,-110.740,61.090,-0.1100,-0.0400,0.9900
C01583=23.570,-115.280,61.750,-0.0900,-0.0700,0.9900
C01584=27.490,-118.440,62.100,-0.0300,-0.0600,1.0000
C01585=32.920,-119.700,62.390,-0.0000,-0.0400,1.0000
C01586=38.860,-118.720,62.680,0.0000,-0.0000,1.0000
C01587=44.850,-116.670,62.870,0.0000,-0.0000,1.0000
C01588=50.780,-114.210,62.870,0.0000,-0.0000,1.0000
C01589=56.470,-111.430,62.680,0.0000,-0.0000,1.0000
C01590=61.360,-107.910,62.390,0.0300,-0.0200,1.0000
C01591=64.320,-103.190,62.100,0.0600,-0.0200,1.0000
C01592=64.850,-98.180,61.750,0.1100,0.0200,0.9900
C01593=63.020,-93.590,61.090,0.1000,0.0500,0.9900
C01594=60.620,-89.000,59.780,0.0600,0.0300,1.0000
C01595=58.580,-84.850,58.090,-0.0200,-0.0100,1.0000
C01596=57.530,-81.360,56.480,-0.2000,-0.0500,0.9800
C01597=58.230,-78.210,55.320,-0.5000,0.2400,0.8300
C01598=61.450,-74.720,54.870,-0.4300,0.4500,0.7800
C01599=65.000,-71.580,54.850,-0.4200,0.4700,0.7800
C01600=68.370,-68.370,54.860,-0.4500,0.4500,0.7800
C01601=71.580,-65.000,54.850,-0.4700,0.4200,0.7800
C01602=74.720,-61.450,54.870,-0.4500,0.4300,0.7800
C01603=78.210,-58.230,55.320,-0.2400,0.5000,0.8300
C01604=81.360,-57.530,56.480,0.0500,0.2000,0.9800
C01605=84.850,-58.580,58.090,0.0100,0.0200,1.0000
C01606=89.000,-60.620,59.780,-0.0300,-0.0600,1.0000
C01607=93.590,-63.020,61.090,-0.0500,-0.1000,0.9900
C01608=98.180,-64.850,61.750,-0.0200,-0.1100,0.9900
C01609=103.190,-64.320,62.100,0.0200,-0.0600,1.0000
C01610=107.910,-61.360,62.390,0.0200,-0.0300,1.0000
C01611=111.430,-56.470,62.680,0.0000,-0.0000,1.0000
C01612=114.210,-50.780,62.870,0.0000,-0.0000,1.0000
C01613=116.670,-44.850,62.870,0.0000,-0.0000,1.0000
C01614=118.720,-38.860,62.680,0.0000,-0.0000,1.0000
C01615=119.700,-32.920,62.390,0.0400,0.0000,1.0000
C01616=118.440,-27.490,62.100,0.0600,0.0300,1.0000
C01617=115.280,-23.570,61.750,0.0700,0.0900,0.9900
C01618=110.740,-21.620,61.090,0.0400,0.1100,0.9900
C01619=105.790,-20.070,59.780,0.0200,0.0700,1.0000
C01620=101.420,-18.580,58.090,-0.0100,-0.0200,1.0000
C01621=98.210,-16.850,56.480,-0.1100,-0.1700,0.9800
C01622=96.480,-14.130,55.320,-0.5300,-0.1800,0.8300
C01623=96.280,-9.390,54.870,-0.6300,0.0100,0.7800
C01624=96.580,-4.650,54.850,-0.6300,0.0300,0.7800
C01625=96.690,0.000,54.860,-0.6300,0.0000,0.7800
C01626=96.580,4.650,54.850,-0.6300,-0.0300,0.7800
C01627=96.280,9.390,54.870,-0.6300,-0.0100,0.7800
C01628=96.480,14.130,55.320,-0.5300,0.1800,0.8300
C01629=98.210,16.850,56.480,-0.1100,0.1700,0.9800
C01630=101.420,18.580,58.090,-0.0100,0.0200,1.0000
C01631=105.790,20.070,59.780,0.0200,-0.0700,1.0000
C01632=110.740,21.620,61.090,0.0400,-0.1100,0.9900
C01633=115.280,23.570,61.750,0.0700,-0.0900,0.9900
C01634=118.440,27.490,62.100,0.0600,-0.0300,1.0000
C01635=119.700,32.920,62.390,0.0400,-0.0000,1.0000
C01636=118.720,38.860,62.680,0.0000,0.0000,1.0000
C01637=116.670,44.850,62.870,0.0000,0.0000,1.0000
C01638=114.210,50.780,62.870,0.0000,0.0000,1.0000
C01639=111.430,56.470,62.680,0.0000,0.0000,1.0000
C01640=107.910,61.360,62.390,0.0200,0.0300,1.0000
C01641=103.190,64.320,62.100,0.0200,0.0600,1.0000
C01642=98.180,64.850,61.750,-0.0200,0.1100,0.9900
C01643=93.590,63.020,61.090,-0.0500,0.1000,0.9900
C01644=89.000,60.620,59.780,-0.0300,0.0600,1.0000
C01645=84.850,58.580,58.090,0.0100,-0.0200,1.0000
C01646=81.360,57.530,56.480,0.0500,-0.2000,0.9800
C01647=78.210,58.230,55.320,-0.2400,-0.5000,0.8300
C01648=74.720,61.450,54.870,-0.4500,-0.4300,0.7800
C01649=71.580,65.000,54.850,-0.4700,-0.4200,0.7800
C01650=68.370,68.370,54.860,-0.4500,-0.4500,0.7800
C01651=65.000,71.580,54.850,-0.4200,-0.4700,0.7800
C01652=61.450,74.720,54.870,-0.4300,-0.4500,0.7800
C01653=58.230,78.210,55.320,-0.5000,-0.2400,0.8300
C01654=57.530,81.360,56.480,-0.2000,0.0500,0.9800
C01655=58.580,84.850,58.090,-0.0200,0.0100,1.0000
C01656=60.620,89.000,59.780,0.0600,-0.0300,1.0000
C01657=63.020,93.590,61.090,0.1000,-0.0500,0.9900
C01658=64.850,98.180,61.750,0.1100,-0.0200,0.9900
C01659=64.320,103.190,62.100,0.0600,0.0200,1.0000
C01660=61.360,107.910,62.390,0.0300,0.0200,1.0000
C01661=56.470,111.430,62.680,0.0000,0.0000,1.0000
C01662=50.780,114.210,62.870,0.0000,0.0000,1.0000
C01663=44.850,116.670,62.870,0.0000,0.0000,1.0000
C01664=38.860,118.720,62.680,0.0000,0.0000,1.0000
C01665=32.920,119.700,62.390,-0.0000,0.0400,1.0000
C01666=27.490,118.440,62.100,-0.0300,0.0600,1.0000
C01667=23.570,115.280,61.750,-0.0900,0.0700,0.9900
C01668=21.620,110.740,61.090,-0.1100,0.0400,0.9900
C01669=20.070,105.790,59.780,-0.0700,0.0200,1.0000
C01670=18.580,101.420,58.090,0.0200,-0.0100,1.0000
C01671=16.850,98.210,56.480,0.1700,-0.1100,0.9800
C01672=14.130,96.480,55.320,0.1800,-0.5300,0.8300
C01673=9.390,96.280,54.870,-0.0100,-0.6300,0.7800
C01674=4.650,96.580,54.850,-0.0300,-0.6300,0.7800
C01675=0.000,96.690,54.860,0.0000,-0.6300,0.7800
C01676=0.000,95.620,56.180,0.0000,-0.6300,0.7800
C01677=4.560,95.510,56.160,-0.0300,-0.6300,0.7800
C01678=9.220,95.230,56.190,-0.0100,-0.6300,0.7800
C01679=13.930,95.450,56.660,0.1900,-0.5200,0.8300
C01680=16.600,97.270,57.870,0.1600,-0.1000,0.9800
C01681=18.290,100.620,59.560,0.0100,-0.0000,1.0000
C01682=19.750,105.170,61.330,-0.0700,0.0200,1.0000
C01683=21.270,110.330,62.710,-0.1100,0.0400,0.9900
C01684=23.190,115.070,63.400,-0.1000,0.0700,0.9900
C01685=27.130,118.400,63.760,-0.0300,0.0600,1.0000
C01686=32.630,119.750,64.070,-0.0000,0.0400,1.0000
C01687=38.690,118.780,64.370,0.0000,0.0000,1.0000
C01688=44.790,116.690,64.570,0.0000,0.0000,1.0000
C01689=50.840,114.180,64.570,0.0000,0.0000,1.0000
C01690=56.630,111.340,64.370,0.0000,0.0000,1.0000
C01691=61.600,107.750,64.070,0.0300,0.0300,1.0000
C01692=64.540,102.900,63.760,0.0700,0.0200,1.0000
C01693=64.970,97.760,63.400,0.1200,-0.0200,0.9900
C01694=62.970,93.050,62.710,0.1100,-0.0500,0.9900
C01695=60.400,88.330,61.330,0.0700,-0.0300,1.0000
C01696=58.210,84.080,59.560,-0.0100,0.0000,1.0000
C01697=57.040,80.520,57.870,-0.1800,0.0500,0.9800
C01698=57.640,77.340,56.660,-0.5000,-0.2300,0.8300
C01699=60.810,73.850,56.190,-0.4400,-0.4500,0.7800
C01700=64.320,70.760,56.160,-0.4200,-0.4700,0.7800
C01701=67.610,67.610,56.180,-0.4500,-0.4500,0.7800
C01702=70.760,64.320,56.160,-0.4700,-0.4200,0.7800
C01703=73.850,60.810,56.190,-0.4500,-0.4400,0.7800
C01704=77.340,57.640,56.660,-0.2300,-0.5000,0.8300
C01705=80.520,57.040,57.870,0.0500,-0.1800,0.9800
C01706=84.080,58.210,59.560,0.0000,-0.0100,1.0000
C01707=88.330,60.400,61.330,-0.0300,0.0700,1.0000
C01708=93.050,62.970,62.710,-0.0500,0.1100,0.9900
C01709=97.760,64.970,63.400,-0.0200,0.1200,0.9900
C01710=102.900,64.540,63.760,0.0200,0.0700,1.0000
C01711=107.750,61.600,64.070,0.0300,0.0300,1.0000
C01712=111.340,56.630,64.370,0.0000,0.0000,1.0000
C01713=114.180,50.840,64.570,0.0000,0.0000,1.0000
C01714=116.690,44.790,64.570,0.0000,0.0000,1.0000
C01715=118.780,38.690,64.370,0.0000,0.0000,1.0000
C01716=119.750,32.630,64.070,0.0400,-0.0000,1.0000
C01717=118.400,27.130,63.760,0.0600,-0.0300,1.0000
C01718=115.070,23.190,63.400,0.0700,-0.1000,0.9900
C01719=110.330,21.270,62.710,0.0400,-0.1100,0.9900
C01720=105.170,19.750,61.330,0.0200,-0.0700,1.0000
C01721=100.620,18.290,59.560,-0.0000,0.0100,1.0000
C01722=97.270,16.600,57.870,-0.1000,0.1600,0.9800
C01723=95.450,13.930,56.660,-0.5200,0.1900,0.8300
C01724=95.230,9.220,56.190,-0.6300,-0.0100,0.7800
C01725=95.510,4.560,56.160,-0.6300,-0.0300,0.7800
C01726=95.620,0.000,56.180,-0.6300,0.0000,0.7800
C01727=95.510,-4.560,56.160,-0.6300,0.0300,0.7800
C01728=95.230,-9.220,56.190,-0.6300,0.0100,0.7800
C01729=95.450,-13.930,56.660,-0.5200,-0.1900,0.8300
C01730=97.270,-16.600,57.870,-0.1000,-0.1600,0.9800
C01731=100.620,-18.290,59.560,-0.0000,-0.0100,1.0000
C01732=105.170,-19.750,61.330,0.0200,0.0700,1.0000
C01733=110.330,-21.270,62.710,0.0400,0.1100,0.9900
C01734=115.070,-23.190,63.400,0.0700,0.1000,0.9900
C01735=118.400,-27.130,63.760,0.0600,0.0300,1.0000
C01736=119.750,-32.630,64.070,0.0400,0.0000,1.0000
C01737=118.780,-38.690,64.370,0.0000,-0.0000,1.0000
C01738=116.690,-44.790,64.570,0.0000,-0.0000,1.0000
C01739=114.180,-50.840,64.570,0.0000,-0.0000,1.0000
C01740=111.340,-56.630,64.370,0.0000,-0.0000,1.0000
C01741=107.750,-61.600,64.070,0.0300,-0.0300,1.0000
C01742=102.900,-64.540,63.760,0.0200,-0.0700,1.0000
C01743=97.760,-64.970,63.400,-0.0200,-0.1200,0.9900
C01744=93.050,-62.970,62.710,-0.0500,-0.1100,0.9900
C01745=88.330,-60.400,61.330,-0.0300,-0.0700,1.0000
C01746=84.080,-58.210,59.560,0.0000,0.0100,1.0000
C01747=80.520,-57.040,57.870,0.0500,0.1800,0.9800
C01748=77.340,-57.640,56.660,-0.2300,0.5000,0.8300
C01749=73.850,-60.810,56.190,-0.4500,0.4400,0.7800
C01750=70.760,-64.320,56.160,-0.4700,0.4200,0.7800
C01751=67.610,-67.610,56.180,-0.4500,0.4500,0.7800
C01752=64.320,-70.760,56.160,-0.4200,0.4700,0.7800
C01753=60.810,-73.850,56.190,-0.4400,0.4500,0.7800
C01754=57.640,-77.340,56.660,-0.5000,0.2300,0.8300
C01755=57.040,-80.520,57.870,-0.1800,-0.0500,0.9800
C01756=58.210,-84.080,59.560,-0.0100,-0.0000,1.0000
C01757=60.400,-88.330,61.330,0.0700,0.0300,1.0000
C01758=62.970,-93.050,62.710,0.1100,0.0500,0.9900
C01759=64.970,-97.760,63.400,0.1200,0.0200,0.9900
C01760=64.540,-102.900,63.760,0.0700,-0.0200,1.0000
C01761=61.600,-107.750,64.070,0.0300,-0.0300,1.0000
C01762=56.630,-111.340,64.370,0.0000,-0.0000,1.0000
C01763=50.840,-114.180,64.570,0.0000,-0.0000,1.0000
C01764=44.790,-116.690,64.570,0.0000,-0.0000,1.0000
C01765=38.690,-118.780,64.370,0.0000,-0.0000,1.0000
C01766=32.630,-119.750,64.070,-0.0000,-0.0400,1.0000
C01767=27.130,-118.400,63.760,-0.0300,-0.0600,1.0000
C01768=23.190,-115.070,63.400,-0.1000,-0.0700,0.9900
C01769=21.270,-110.330,62.710,-0.1100,-0.0400,0.9900
C01770=19.750,-105.170,61.330,-0.0700,-0.0200,1.0000
C01771=18.290,-100.620,59.560,0.0100,0.0000,1.0000
C01772=16.600,-97.270,57.870,0.1600,0.1000,0.9800
C01773=13.930,-95.450,56.660,0.1900,0.5200,0.8300
C01774=9.220,-95.230,56.190,-0.0100,0.6300,0.7800
C01775=4.560,-95.510,56.160,-0.0300,0.6300,0.7800
C01776=0.000,-95.620,56.180,0.0000,0.6300,0.7800
C01777=0.000,-95.620,56.180,0.0000,0.6300,0.7800
C01778=-4.560,-95.510,56.160,0.0300,0.6300,0.7800
C01779=-9.220,-95.230,56.190,0.0100,0.6300,0.7800
C01780=-13.930,-95.450,56.660,-0.1900,0.5200,0.8300
C01781=-16.600,-97.270,57.870,-0.1600,0.1000,0.9800
C01782=-18.290,-100.620,59.560,-0.0100,0.0000,1.0000
C01783=-19.750,-105.170,61.330,0.0700,-0.0200,1.0000
C01784=-21.270,-110.330,62.710,0.1100,-0.0400,0.9900
C01785=-23.190,-115.070,63.400,0.1000,-0.0700,0.9900
C01786=-27.130,-118.400,63.760,0.0300,-0.0600,1.0000
C01787=-32.630,-119.750,64.070,0.0000,-0.0400,1.0000
C01788=-38.690,-118.780,64.370,-0.0000,-0.0000,1.0000
C01789=-44.790,-116.690,64.570,-0.0000,-0.0000,1.0000
C01790=-50.840,-114.180,64.570,-0.0000,-0.0000,1.0000
C01791=-56.630,-111.340,64.370,-0.0000,-0.0000,1.0000
C01792=-61.600,-107.750,64.070,-0.0300,-0.0300,1.0000
C01793=-64.540,-102.900,63.760,-0.0700,-0.0200,1.0000
C01794=-64.970,-97.760,63.400,-0.1200,0.0200,0.9900
C01795=-62.970,-93.050,62.710,-0.1100,0.0500,0.9900
C01796=-60.400,-88.330,61.330,-0.0700,0.0300,1.0000
C01797=-58.210,-84.080,59.560,0.0100,-0.0000,1.0000
C01798=-57.040,-80.520,57.870,0.1800,-0.0500,0.9800
C01799=-57.640,-77.340,56.660,0.5000,0.2300,0.8300
C01800=-60.810,-73.850,56.190,0.4400,0.4500,0.7800
C01801=-64.320,-70.760,56.160,0.4200,0.4700,0.7800
C01802=-67.610,-67.610,56.180,0.4500,0.4500,0.7800
C01803=-70.760,-64.320,56.160,0.4700,0.4200,0.7800
C01804=-73.850,-60.810,56.190,0.4500,0.4400,0.7800
C01805=-77.340,-57.640,56.660,0.2300,0.5000,0.8300
C01806=-80.520,-57.040,57.870,-0.0500,0.1800,0.9800
C01807=-84.080,-58.210,59.560,-0.0000,0.0100,1.0000
C01808=-88.330,-60.400,61.330,0.0300,-0.0700,1.0000
C01809=-93.050,-62.970,62.710,0.0500,-0.1100,0.9900
C01810=-97.760,-64.970,63.400,0.0200,-0.1200,0.9900
C01811=-102.900,-64.540,63.760,-0.0200,-0.0700,1.0000
C01812=-107.750,-61.600,64.070,-0.0300,-0.0300,1.0000
C01813=-111.340,-56.630,64.370,-0.0000,-0.0000,1.0000
C01814=-114.180,-50.840,64.570,-0.0000,-0.0000,1.0000
C01815=-116.690,-44.790,64.570,-0.0000,-0.0000,1.0000
C01816=-118.780,-38.690,64.370,-0.0000,-0.0000,1.0000
C01817=-119.750,-32.630,64.070,-0.0400,0.0000,1.0000
C01818=-118.400,-27.130,63.760,-0.0600,0.0300,1.0000
C01819=-115.070,-23.190,63.400,-0.0700,0.1000,0.9900
C01820=-110.330,-21.270,62.710,-0.0400,0.1100,0.9900
C01821=-105.170,-19.750,61.330,-0.0200,0.0700,1.0000
C01822=-100.620,-18.290,59.560,0.0000,-0.0100,1.0000
C01823=-97.270,-16.600,57.870,0.1000,-0.1600,0.9800
C01824=-95.450,-13.930,56.660,0.5200,-0.1900,0.8300
C01825=-95.230,-9.220,56.190,0.6300,0.0100,0.7800
C01826=-95.510,-4.560,56.160,0.6300,0.0300,0.7800
C01827=-95.620,0.000,56.180,0.6300,-0.0000,0.7800
C01828=-95.510,4.560,56.160,0.6300,-0.0300,0.7800
C01829=-95.230,9.220,56.190,0.6300,-0.0100,0.7800
C01830=-95.450,13.930,56.660,0.5200,0.1900,0.8300
C01831=-97.270,16.600,57.870,0.1000,0.1600,0.9800
C01832=-100.620,18.290,59.560,0.0000,0.0100,1.0000
C01833=-105.170,19.750,61.330,-0.0200,-0.0700,1.0000
C01834=-110.330,21.270,62.710,-0.0400,-0.1100,0.9900
C01835=-115.070,23.190,63.400,-0.0700,-0.1000,0.9900
C01836=-118.400,27.130,63.760,-0.0600,-0.0300,1.0000
C01837=-119.750,32.630,64.070,-0.0400,-0.0000,1.0000
C01838=-118.780,38.690,64.370,-0.0000,0.0000,1.0000
C01839=-116.690,44.790,64.570,-0.0000,0.0000,1.0000
C01840=-114.180,50.840,64.570,-0.0000,0.0000,1.0000
C01841=-111.340,56.630,64.370,-0.0000,0.0000,1.0000
C01842=-107.750,61.600,64.070,-0.0300,0.0300,1.0000
C01843=-102.900,64.540,63.760,-0.0200,0.0700,1.0000
C01844=-97.760,64.970,63.400,0.0200,0.1200,0.9900
C01845=-93.050,62.970,62.710,0.0500,0.1100,0.9900
C01846=-88.330,60.400,61.330,0.0300,0.0700,1.0000
C01847=-84.080,58.210,59.560,-0.0000,-0.0100,1.0000
C01848=-80.520,57.040,57.870,-0.0500,-0.1800,0.9800
C01849=-77.340,57.640,56.660,0.2300,-0.5000,0.8300
C01850=-73.850,60.810,56.190,0.4500,-0.4400,0.7800
C01851=-70.760,64.320,56.160,0.4700,-0.4200,0.7800
C01852=-67.610,67.610,56.180,0.4500,-0.4500,0.7800
C01853=-64.320,70.760,56.160,0.4200,-0.4700,0.7800
C01854=-60.810,73.850,56.190,0.4400,-0.4500,0.7800
C01855=-57.640,77.340,56.660,0.5000,-0.2300,0.8300
C01856=-57.040,80.520,57.870,0.1800,0.0500,0.9800
C01857=-58.210,84.080,59.560,0.0100,0.0000,1.0000
C01858=-60.400,88.330,61.330,-0.0700,-0.0300,1.0000
C01859=-62.970,93.050,62.710,-0.1100,-0.0500,0.9900
C01860=-64.970,97.760,63.400,-0.1200,-0.0200,0.9900
C01861=-64.540,102.900,63.760,-0.0700,0.0200,1.0000
C01862=-61.600,107.750,64.070,-0.0300,0.0300,1.0000
C01863=-56.630,111.340,64.370,-0.0000,0.0000,1.0000
C01864=-50.840,114.180,64.570,-0.0000,0.0000,1.0000
C01865=-44.790,116.690,64.570,-0.0000,0.0000,1.0000
C01866=-38.690,118.780,64.370,-0.0000,0.0000,1.0000
C01867=-32.630,119.750,64.070,0.0000,0.0400,1.0000
C01868=-27.130,118.400,63.760,0.0300,0.0600,1.0000
C01869=-23.190,115.070,63.400,0.1000,0.0700,0.9900
C01870=-21.270,110.330,62.710,0.1100,0.0400,0.9900
C01871=-19.750,105.170,61.330,0.0700,0.0200,1.0000
C01872=-18.290,100.620,59.560,-0.0100,-0.0000,1.0000
C01873=-16.600,97.270,57.870,-0.1600,-0.1000,0.9800
C01874=-13.930,95.450,56.660,-0.1900,-0.5200,0.8300
C01875=-9.220,95.230,56.190,0.0100,-0.6300,0.7800
C01876=-4.560,95.510,56.160,0.0300,-0.6300,0.7800
C01877=0.000,95.620,56.180,0.0000,-0.6300,0.7800
C01878=0.000,94.550,57.500,0.0000,-0.6300,0.7700
C01879=-4.460,94.440,57.480,0.0300,-0.6300,0.7700
C01880=-9.060,94.160,57.500,0.0100,-0.6300,0.7800
C01881=-13.720,94.420,58.000,-0.2000,-0.5100,0.8300
C01882=-16.350,96.330,59.270,-0.1500,-0.0800,0.9800
C01883=-18.000,99.810,61.030,0.0000,0.0000,1.0000
C01884=-19.430,104.550,62.880,0.0800,0.0200,1.0000
C01885=-20.930,109.910,64.320,0.1200,0.0400,0.9900
C01886=-22.810,114.870,65.040,0.1000,0.0700,0.9900
C01887=-26.770,118.360,65.430,0.0300,0.0700,1.0000
C01888=-32.350,119.800,65.740,0.0000,0.0400,1.0000
C01889=-38.510,118.840,66.060,-0.0000,0.0000,1.0000
C01890=-44.730,116.710,66.270,-0.0000,0.0000,1.0000
C01891=-50.900,114.160,66.270,-0.0000,0.0000,1.0000
C01892=-56.800,111.260,66.060,-0.0000,0.0000,1.0000
C01893=-61.840,107.590,65.740,-0.0300,0.0300,1.0000
C01894=-64.760,102.620,65.430,-0.0700,0.0200,1.0000
C01895=-65.090,97.350,65.040,-0.1200,-0.0300,0.9900
C01896=-62.920,92.520,64.320,-0.1100,-0.0600,0.9900
C01897=-60.190,87.670,62.880,-0.0700,-0.0400,1.0000
C01898=-57.850,83.300,61.030,-0.0000,-0.0000,1.0000
C01899=-56.550,79.670,59.270,0.1700,0.0500,0.9800
C01900=-57.060,76.470,58.000,0.5100,-0.2200,0.8300
C01901=-60.180,72.990,57.500,0.4400,-0.4500,0.7800
C01902=-63.630,69.930,57.480,0.4200,-0.4700,0.7700
C01903=-66.860,66.860,57.500,0.4500,-0.4500,0.7700
C01904=-69.930,63.630,57.480,0.4700,-0.4200,0.7700
C01905=-72.990,60.180,57.500,0.4500,-0.4400,0.7800
C01906=-76.470,57.060,58.000,0.2200,-0.5100,0.8300
C01907=-79.670,56.550,59.270,-0.0500,-0.1700,0.9800
C01908=-83.300,57.850,61.030,0.0000,0.0000,1.0000
C01909=-87.670,60.190,62.880,0.0400,0.0700,1.0000
C01910=-92.520,62.920,64.320,0.0600,0.1100,0.9900
C01911=-97.350,65.090,65.040,0.0300,0.1200,0.9900
C01912=-102.620,64.760,65.430,-0.0200,0.0700,1.0000
C01913=-107.590,61.840,65.740,-0.0300,0.0300,1.0000
C01914=-111.260,56.800,66.060,-0.0000,0.0000,1.0000
C01915=-114.160,50.900,66.270,-0.0000,0.0000,1.0000
C01916=-116.710,44.730,66.270,-0.0000,0.0000,1.0000
C01917=-118.840,38.510,66.060,-0.0000,0.0000,1.0000
C01918=-119.800,32.350,65.740,-0.0400,-0.0000,1.0000
C01919=-118.360,26.770,65.430,-0.0700,-0.0300,1.0000
C01920=-114.870,22.810,65.040,-0.0700,-0.1000,0.9900
C01921=-109.910,20.930,64.320,-0.0400,-0.1200,0.9900
C01922=-104.550,19.430,62.880,-0.0200,-0.0800,1.0000
C01923=-99.810,18.000,61.030,-0.0000,-0.0000,1.0000
C01924=-96.330,16.350,59.270,0.0800,0.1500,0.9800
C01925=-94.420,13.720,58.000,0.5100,0.2000,0.8300
C01926=-94.160,9.060,57.500,0.6300,-0.0100,0.7800
C01927=-94.440,4.460,57.480,0.6300,-0.0300,0.7700
C01928=-94.550,0.000,57.500,0.6300,-0.0000,0.7700
C01929=-94.440,-4.460,57.480,0.6300,0.0300,0.7700
C01930=-94.160,-9.060,57.500,0.6300,0.0100,0.7800
C01931=-94.420,-13.720,58.000,0.5100,-0.2000,0.8300
C01932=-96.330,-16.350,59.270,0.0800,-0.1500,0.9800
C01933=-99.810,-18.000,61.030,-0.0000,0.0000,1.0000
C01934=-104.550,-19.430,62.880,-0.0200,0.0800,1.0000
C01935=-109.910,-20.930,64.320,-0.0400,0.1200,0.9900
